LIN {X 6.039,Y -16.044,Z -36.377,A -90.000,B 90.000,C 0.000} C_DIS
LIN {X 6.734,Y -16.027,Z -36.490,A -90.000,B 90.000,C 0.000} C_DIS
LIN {X 7.092,Y -16.027,Z -36.557,A -90.000,B 90.000,C 0.000} C_DIS
LIN {X 7.740,Y -16.017,Z -36.687,A -90.000,B 90.000,C 0.000} C_DIS
LIN {X 9.449,Y -15.968,Z -37.009,A -90.000,B 90.000,C 0.000} C_DIS
LIN {X 9.774,Y -15.964,Z -37.078,A -90.000,B 90.000,C 0.000} C_DIS
LIN {X 10.396,Y -15.956,Z -37.212,A -90.000,B 90.000,C 0.000} C_DIS
LIN {X 11.916,Y -15.912,Z -37.509,A -90.000,B 90.000,C 0.000} C_DIS
LIN {X 12.481,Y -15.903,Z -37.625,A -90.000,B 90.000,C 0.000} C_DIS
LIN {X 13.325,Y -15.897,Z -37.792,A -90.000,B 90.000,C 0.000} C_DIS
LIN {X 14.273,Y -15.872,Z -37.963,A -90.000,B 90.000,C 0.000} C_DIS
LIN {X 14.869,Y -15.862,Z -38.055,A -90.000,B 90.000,C 0.000} C_DIS
LIN {X 16.056,Y -15.855,Z -38.223,A -90.000,B 90.000,C 0.000} C_DIS
LIN {X 16.523,Y -15.850,Z -38.287,A -90.000,B 90.000,C 0.000} C_DIS
LIN {X 16.570,Y -15.848,Z -38.291,A -90.000,B 90.000,C 0.000} C_DIS
LIN {X 16.973,Y -15.845,Z -38.311,A -90.000,B 90.000,C 0.000} C_DIS
LIN {X 17.413,Y -15.859,Z -38.314,A -90.000,B 90.000,C 0.000} C_DIS
LIN {X 18.246,Y -15.862,Z -38.297,A -90.000,B 90.000,C 0.000} C_DIS
LIN {X 19.359,Y -15.901,Z -38.239,A -90.000,B 90.000,C 0.000} C_DIS
LIN {X 20.076,Y -15.912,Z -38.189,A -90.000,B 90.000,C 0.000} C_DIS
LIN {X 20.520,Y -15.912,Z -38.152,A -90.000,B 90.000,C 0.000} C_DIS
LIN {X 21.087,Y -15.918,Z -38.097,A -90.000,B 90.000,C 0.000} C_DIS
LIN {X 21.632,Y -15.923,Z -38.047,A -90.000,B 90.000,C 0.000} C_DIS
LIN {X 22.818,Y -15.923,Z -37.927,A -90.000,B 90.000,C 0.000} C_DIS
LIN {X 23.377,Y -15.913,Z -37.881,A -90.000,B 90.000,C 0.000} C_DIS
LIN {X 23.875,Y -15.906,Z -37.843,A -90.000,B 90.000,C 0.000} C_DIS
LIN {X 24.231,Y -15.897,Z -37.817,A -90.000,B 90.000,C 0.000} C_DIS
LIN {X 24.592,Y -15.885,Z -37.793,A -90.000,B 90.000,C 0.000} C_DIS
LIN {X 25.132,Y -15.871,Z -37.753,A -90.000,B 90.000,C 0.000} C_DIS
LIN {X 26.019,Y -15.831,Z -37.672,A -90.000,B 90.000,C 0.000} C_DIS
LIN {X 26.243,Y -15.824,Z -37.649,A -90.000,B 90.000,C 0.000} C_DIS
LIN {X 26.557,Y -15.821,Z -37.620,A -90.000,B 90.000,C 0.000} C_DIS
LIN {X 26.906,Y -15.809,Z -37.600,A -90.000,B 90.000,C 0.000} C_DIS
LIN {X 27.052,Y -15.798,Z -37.586,A -90.000,B 90.000,C 0.000} C_DIS
LIN {X 27.543,Y -15.770,Z -37.548,A -90.000,B 90.000,C 0.000} C_DIS
LIN {X 27.884,Y -15.754,Z -37.527,A -90.000,B 90.000,C 0.000} C_DIS
LIN {X 28.286,Y -15.743,Z -37.494,A -90.000,B 90.000,C 0.000} C_DIS
LIN {X 28.880,Y -15.723,Z -37.457,A -90.000,B 90.000,C 0.000} C_DIS
LIN {X 29.189,Y -15.702,Z -37.445,A -90.000,B 90.000,C 0.000} C_DIS
LIN {X 29.939,Y -15.655,Z -37.419,A -90.000,B 90.000,C 0.000} C_DIS
LIN {X 30.142,Y -15.646,Z -37.409,A -90.000,B 90.000,C 0.000} C_DIS
LIN {X 30.320,Y -15.634,Z -37.406,A -90.000,B 90.000,C 0.000} C_DIS
LIN {X 30.803,Y -15.614,Z -37.401,A -90.000,B 90.000,C 0.000} C_DIS
LIN {X 31.147,Y -15.605,Z -37.400,A -90.000,B 90.000,C 0.000} C_DIS
LIN {X 31.402,Y -15.589,Z -37.395,A -90.000,B 90.000,C 0.000} C_DIS
LIN {X 32.076,Y -15.550,Z -37.383,A -90.000,B 90.000,C 0.000} C_DIS
LIN {X 32.349,Y -15.534,Z -37.383,A -90.000,B 90.000,C 0.000} C_DIS
LIN {X 33.413,Y -15.503,Z -37.403,A -90.000,B 90.000,C 0.000} C_DIS
LIN {X 33.723,Y -15.486,Z -37.406,A -90.000,B 90.000,C 0.000} C_DIS
LIN {X 34.278,Y -15.462,Z -37.418,A -90.000,B 90.000,C 0.000} C_DIS
LIN {X 34.543,Y -15.456,Z -37.421,A -90.000,B 90.000,C 0.000} C_DIS
LIN {X 34.797,Y -15.450,Z -37.428,A -90.000,B 90.000,C 0.000} C_DIS
LIN {X 35.524,Y -15.428,Z -37.462,A -90.000,B 90.000,C 0.000} C_DIS
LIN {X 36.099,Y -15.416,Z -37.491,A -90.000,B 90.000,C 0.000} C_DIS
LIN {X 36.763,Y -15.397,Z -37.551,A -90.000,B 90.000,C 0.000} C_DIS
LIN {X 37.410,Y -15.387,Z -37.613,A -90.000,B 90.000,C 0.000} C_DIS
LIN {X 37.906,Y -15.374,Z -37.682,A -90.000,B 90.000,C 0.000} C_DIS
LIN {X 38.646,Y -15.360,Z -37.787,A -90.000,B 90.000,C 0.000} C_DIS
LIN {X 39.682,Y -15.341,Z -37.952,A -90.000,B 90.000,C 0.000} C_DIS
LIN {X 40.000,Y -15.341,Z -38.004,A -90.000,B 90.000,C 0.000} C_DIS
LIN {X 40.509,Y -15.338,Z -38.097,A -90.000,B 90.000,C 0.000} C_DIS
LIN {X 41.041,Y -15.331,Z -38.226,A -90.000,B 90.000,C 0.000} C_DIS
LIN {X 42.380,Y -15.317,Z -38.551,A -90.000,B 90.000,C 0.000} C_DIS
LIN {X 43.069,Y -15.313,Z -38.719,A -90.000,B 90.000,C 0.000} C_DIS
LIN {X 43.342,Y -15.313,Z -38.782,A -90.000,B 90.000,C 0.000} C_DIS
LIN {X 43.874,Y -15.312,Z -38.938,A -90.000,B 90.000,C 0.000} C_DIS
LIN {X 45.211,Y -15.309,Z -39.381,A -90.000,B 90.000,C 0.000} C_DIS
LIN {X 46.407,Y -15.308,Z -39.801,A -90.000,B 90.000,C 0.000} C_DIS
LIN {X 46.548,Y -15.315,Z -39.851,A -90.000,B 90.000,C 0.000} C_DIS
LIN {X 46.604,Y -15.308,Z -39.871,A -90.000,B 90.000,C 0.000} C_DIS
LIN {X 47.058,Y -15.309,Z -40.058,A -90.000,B 90.000,C 0.000} C_DIS
LIN {X 49.401,Y -15.308,Z -41.077,A -90.000,B 90.000,C 0.000} C_DIS
LIN {X 49.533,Y -15.308,Z -41.134,A -90.000,B 90.000,C 0.000} C_DIS
LIN {X 49.660,Y -15.308,Z -41.203,A -90.000,B 90.000,C 0.000} C_DIS
LIN {X 49.716,Y -15.308,Z -41.231,A -90.000,B 90.000,C 0.000} C_DIS
LIN {X 50.779,Y -15.308,Z -41.767,A -90.000,B 90.000,C 0.000} C_DIS
LIN {X 51.050,Y -15.308,Z -41.899,A -90.000,B 90.000,C 0.000} C_DIS
LIN {X 51.127,Y -15.308,Z -41.932,A -90.000,B 90.000,C 0.000} C_DIS
LIN {X 51.197,Y -15.308,Z -41.976,A -90.000,B 90.000,C 0.000} C_DIS
LIN {X 51.458,Y -15.308,Z -42.127,A -90.000,B 90.000,C 0.000} C_DIS
LIN {X 52.496,Y -15.308,Z -42.710,A -90.000,B 90.000,C 0.000} C_DIS
LIN {X 52.552,Y -15.308,Z -42.742,A -90.000,B 90.000,C 0.000} C_DIS
LIN {X 53.714,Y -15.307,Z -43.381,A -90.000,B 90.000,C 0.000} C_DIS
LIN {X 54.187,Y -15.306,Z -43.636,A -90.000,B 90.000,C 0.000} C_DIS
LIN {X 54.943,Y -15.302,Z -44.031,A -90.000,B 90.000,C 0.000} C_DIS
LIN {X 55.235,Y -15.300,Z -44.179,A -90.000,B 90.000,C 0.000} C_DIS
LIN {X 55.671,Y -15.295,Z -44.390,A -90.000,B 90.000,C 0.000} C_DIS
LIN {X 56.151,Y -15.273,Z -44.596,A -90.000,B 90.000,C 0.000} C_DIS
LIN {X 56.148,Y -15.270,Z -44.610,A -90.000,B 90.000,C 0.000} C_DIS
LIN {X 56.151,Y -15.268,Z -44.630,A -90.000,B 90.000,C 0.000} C_DIS
LIN {X 56.175,Y -15.267,Z -44.683,A -90.000,B 90.000,C 0.000} C_DIS
LIN {X 56.236,Y -15.266,Z -44.775,A -90.000,B 90.000,C 0.000} C_DIS
LIN {X 56.306,Y -15.267,Z -44.862,A -90.000,B 90.000,C 0.000} C_DIS
LIN {X 56.404,Y -15.268,Z -44.975,A -90.000,B 90.000,C 0.000} C_DIS
LIN {X 56.536,Y -15.269,Z -45.116,A -90.000,B 90.000,C 0.000} C_DIS
LIN {X 56.707,Y -15.272,Z -45.288,A -90.000,B 90.000,C 0.000} C_DIS
LIN {X 56.921,Y -15.275,Z -45.496,A -90.000,B 90.000,C 0.000} C_DIS
LIN {X 57.333,Y -15.281,Z -45.880,A -90.000,B 90.000,C 0.000} C_DIS
LIN {X 57.870,Y -15.289,Z -46.362,A -90.000,B 90.000,C 0.000} C_DIS
LIN {X 58.080,Y -15.293,Z -46.546,A -90.000,B 90.000,C 0.000} C_DIS
LIN {X 58.309,Y -15.296,Z -46.738,A -90.000,B 90.000,C 0.000} C_DIS
LIN {X 58.812,Y -15.304,Z -47.169,A -90.000,B 90.000,C 0.000} C_DIS
LIN {X 59.086,Y -15.308,Z -47.410,A -90.000,B 90.000,C 0.000} C_DIS
LIN {X 59.874,Y -15.321,Z -48.077,A -90.000,B 90.000,C 0.000} C_DIS
LIN {X 59.965,Y -15.308,Z -48.154,A -90.000,B 90.000,C 0.000} C_DIS
LIN {X 60.154,Y -18.803,Z -48.315,A -90.000,B 90.000,C 0.000} C_DIS
LIN {X 60.177,Y -18.801,Z -48.335,A -90.000,B 90.000,C 0.000} C_DIS
LIN {X 60.181,Y -18.797,Z -48.338,A -90.000,B 90.000,C 0.000} C_DIS
LIN {X 60.185,Y -18.774,Z -48.340,A -90.000,B 90.000,C 0.000} C_DIS
LIN {X 60.211,Y -18.708,Z -48.359,A -90.000,B 90.000,C 0.000} C_DIS
LIN {X 60.278,Y -18.515,Z -48.410,A -90.000,B 90.000,C 0.000} C_DIS
LIN {X 60.408,Y -15.308,Z -48.512,A -90.000,B 90.000,C 0.000} C_DIS
LIN {X 61.034,Y -15.309,Z -49.006,A -90.000,B 90.000,C 0.000} C_DIS
LIN {X 61.707,Y -15.310,Z -49.496,A -90.000,B 90.000,C 0.000} C_DIS
LIN {X 62.539,Y -15.313,Z -50.057,A -90.000,B 90.000,C 0.000} C_DIS
LIN {X 63.422,Y -15.320,Z -50.613,A -90.000,B 90.000,C 0.000} C_DIS
LIN {X 63.809,Y -15.325,Z -50.838,A -90.000,B 90.000,C 0.000} C_DIS
LIN {X 64.774,Y -15.332,Z -51.402,A -90.000,B 90.000,C 0.000} C_DIS
LIN {X 65.381,Y -15.337,Z -51.760,A -90.000,B 90.000,C 0.000} C_DIS
LIN {X 65.866,Y -15.341,Z -52.028,A -90.000,B 90.000,C 0.000} C_DIS
LIN {X 66.964,Y -15.343,Z -52.631,A -90.000,B 90.000,C 0.000} C_DIS
LIN {X 67.835,Y -15.347,Z -53.100,A -90.000,B 90.000,C 0.000} C_DIS
LIN {X 70.105,Y -15.348,Z -54.375,A -90.000,B 90.000,C 0.000} C_DIS
LIN {X 72.147,Y -15.347,Z -55.600,A -90.000,B 90.000,C 0.000} C_DIS
LIN {X 72.312,Y -15.348,Z -55.699,A -90.000,B 90.000,C 0.000} C_DIS
LIN {X 74.555,Y -15.349,Z -57.175,A -90.000,B 90.000,C 0.000} C_DIS
LIN {X 74.781,Y -15.352,Z -57.328,A -90.000,B 90.000,C 0.000} C_DIS
LIN {X 75.952,Y -15.356,Z -58.195,A -90.000,B 90.000,C 0.000} C_DIS
LIN {X 76.534,Y -15.359,Z -58.633,A -90.000,B 90.000,C 0.000} C_DIS
LIN {X 76.658,Y -15.359,Z -58.736,A -90.000,B 90.000,C 0.000} C_DIS
LIN {X 77.528,Y -15.366,Z -59.460,A -90.000,B 90.000,C 0.000} C_DIS
LIN {X 78.045,Y -15.370,Z -59.891,A -90.000,B 90.000,C 0.000} C_DIS
LIN {X 78.182,Y -15.370,Z -60.009,A -90.000,B 90.000,C 0.000} C_DIS
LIN {X 78.182,Y -60.000,Z -60.009,A -90.000,B 90.000,C 0.000} C_DIS
LIN {X 98.807,Y -60.000,Z -39.522,A -90.000,B 90.000,C 0.000} C_DIS
LIN {X 98.807,Y -15.308,Z -39.522,A -90.000,B 90.000,C 0.000} C_DIS
LIN {X 98.954,Y -15.308,Z -39.452,A -90.000,B 90.000,C 0.000} C_DIS
LIN {X 98.954,Y -60.000,Z -39.452,A -90.000,B 90.000,C 0.000} C_DIS
LIN {X 117.188,Y -60.000,Z -45.983,A -90.000,B 90.000,C 0.000} C_DIS
LIN {X 117.188,Y -15.308,Z -45.983,A -90.000,B 90.000,C 0.000} C_DIS
LIN {X 117.180,Y -15.308,Z -46.008,A -90.000,B 90.000,C 0.000} C_DIS
LIN {X 117.180,Y -60.000,Z -46.008,A -90.000,B 90.000,C 0.000} C_DIS
LIN {X -92.086,Y -60.000,Z -21.753,A -90.000,B 90.000,C 0.000} C_DIS
LIN {X -92.086,Y -15.308,Z -21.753,A -90.000,B 90.000,C 0.000} C_DIS
LIN {X -91.888,Y -15.383,Z -21.822,A -90.000,B 90.000,C 0.000} C_DIS
LIN {X -91.713,Y -15.437,Z -21.889,A -90.000,B 90.000,C 0.000} C_DIS
LIN {X -91.547,Y -15.487,Z -21.957,A -90.000,B 90.000,C 0.000} C_DIS
LIN {X -91.432,Y -15.522,Z -22.009,A -90.000,B 90.000,C 0.000} C_DIS
LIN {X -91.308,Y -15.555,Z -22.068,A -90.000,B 90.000,C 0.000} C_DIS
LIN {X -91.116,Y -15.602,Z -22.162,A -90.000,B 90.000,C 0.000} C_DIS
LIN {X -90.998,Y -15.635,Z -22.071,A -90.000,B 90.000,C 0.000} C_DIS
LIN {X -90.915,Y -15.658,Z -22.014,A -90.000,B 90.000,C 0.000} C_DIS
LIN {X -90.848,Y -15.675,Z -21.973,A -90.000,B 90.000,C 0.000} C_DIS
LIN {X -90.705,Y -15.711,Z -21.896,A -90.000,B 90.000,C 0.000} C_DIS
LIN {X -90.601,Y -15.737,Z -21.846,A -90.000,B 90.000,C 0.000} C_DIS
LIN {X -90.508,Y -15.760,Z -21.795,A -90.000,B 90.000,C 0.000} C_DIS
LIN {X -90.443,Y -15.772,Z -21.761,A -90.000,B 90.000,C 0.000} C_DIS
LIN {X -90.207,Y -15.808,Z -21.626,A -90.000,B 90.000,C 0.000} C_DIS
LIN {X -89.996,Y -15.833,Z -21.517,A -90.000,B 90.000,C 0.000} C_DIS
LIN {X -89.781,Y -15.852,Z -21.411,A -90.000,B 90.000,C 0.000} C_DIS
LIN {X -89.618,Y -15.868,Z -21.338,A -90.000,B 90.000,C 0.000} C_DIS
LIN {X -89.570,Y -15.872,Z -21.314,A -90.000,B 90.000,C 0.000} C_DIS
LIN {X -89.396,Y -15.862,Z -21.035,A -90.000,B 90.000,C 0.000} C_DIS
LIN {X -89.237,Y -15.854,Z -20.805,A -90.000,B 90.000,C 0.000} C_DIS
LIN {X -89.137,Y -15.841,Z -20.666,A -90.000,B 90.000,C 0.000} C_DIS
LIN {X -89.073,Y -15.829,Z -20.580,A -90.000,B 90.000,C 0.000} C_DIS
LIN {X -88.905,Y -15.795,Z -20.375,A -90.000,B 90.000,C 0.000} C_DIS
LIN {X -88.721,Y -15.747,Z -20.158,A -90.000,B 90.000,C 0.000} C_DIS
LIN {X -88.629,Y -15.719,Z -20.052,A -90.000,B 90.000,C 0.000} C_DIS
LIN {X -88.477,Y -15.662,Z -19.900,A -90.000,B 90.000,C 0.000} C_DIS
LIN {X -88.436,Y -15.647,Z -19.862,A -90.000,B 90.000,C 0.000} C_DIS
LIN {X -88.404,Y -15.624,Z -19.807,A -90.000,B 90.000,C 0.000} C_DIS
LIN {X -88.259,Y -15.535,Z -19.590,A -90.000,B 90.000,C 0.000} C_DIS
LIN {X -88.129,Y -15.439,Z -19.413,A -90.000,B 90.000,C 0.000} C_DIS
LIN {X -88.068,Y -15.399,Z -19.336,A -90.000,B 90.000,C 0.000} C_DIS
LIN {X -87.988,Y -15.346,Z -19.237,A -90.000,B 90.000,C 0.000} C_DIS
LIN {X -87.929,Y -15.308,Z -19.168,A -90.000,B 90.000,C 0.000} C_DIS
LIN {X -87.929,Y -60.000,Z -19.168,A -90.000,B 90.000,C 0.000} C_DIS
LIN {X -116.648,Y -60.000,Z -243.561,A -90.000,B 90.000,C 0.000} C_DIS
LIN {X -116.648,Y -15.666,Z -243.561,A -90.000,B 90.000,C 0.000} C_DIS
LIN {X -116.613,Y -15.603,Z -243.444,A -90.000,B 90.000,C 0.000} C_DIS
LIN {X -116.514,Y -15.450,Z -243.147,A -90.000,B 90.000,C 0.000} C_DIS
LIN {X -116.456,Y -15.375,Z -242.994,A -90.000,B 90.000,C 0.000} C_DIS
LIN {X -116.391,Y -15.308,Z -242.850,A -90.000,B 90.000,C 0.000} C_DIS
LIN {X -116.376,Y -15.293,Z -242.802,A -90.000,B 90.000,C 0.000} C_DIS
LIN {X -116.360,Y -15.273,Z -242.761,A -90.000,B 90.000,C 0.000} C_DIS
LIN {X -116.349,Y -15.254,Z -242.726,A -90.000,B 90.000,C 0.000} C_DIS
LIN {X -116.337,Y -15.221,Z -242.668,A -90.000,B 90.000,C 0.000} C_DIS
LIN {X -116.338,Y -15.193,Z -242.628,A -90.000,B 90.000,C 0.000} C_DIS
LIN {X -116.342,Y -15.182,Z -242.614,A -90.000,B 90.000,C 0.000} C_DIS
LIN {X -116.361,Y -15.161,Z -242.597,A -90.000,B 90.000,C 0.000} C_DIS
LIN {X -116.382,Y -15.146,Z -242.590,A -90.000,B 90.000,C 0.000} C_DIS
LIN {X -116.419,Y -15.130,Z -242.593,A -90.000,B 90.000,C 0.000} C_DIS
LIN {X -116.466,Y -15.118,Z -242.609,A -90.000,B 90.000,C 0.000} C_DIS
LIN {X -116.522,Y -15.110,Z -242.637,A -90.000,B 90.000,C 0.000} C_DIS
LIN {X -116.586,Y -15.105,Z -242.674,A -90.000,B 90.000,C 0.000} C_DIS
LIN {X -116.692,Y -15.103,Z -242.747,A -90.000,B 90.000,C 0.000} C_DIS
LIN {X -116.768,Y -15.105,Z -242.805,A -90.000,B 90.000,C 0.000} C_DIS
LIN {X -116.929,Y -15.117,Z -242.937,A -90.000,B 90.000,C 0.000} C_DIS
LIN {X -117.012,Y -15.126,Z -243.008,A -90.000,B 90.000,C 0.000} C_DIS
LIN {X -117.174,Y -15.148,Z -243.157,A -90.000,B 90.000,C 0.000} C_DIS
LIN {X -117.251,Y -15.161,Z -243.231,A -90.000,B 90.000,C 0.000} C_DIS
LIN {X -117.393,Y -15.189,Z -243.374,A -90.000,B 90.000,C 0.000} C_DIS
LIN {X -117.510,Y -15.218,Z -243.501,A -90.000,B 90.000,C 0.000} C_DIS
LIN {X -117.557,Y -15.233,Z -243.555,A -90.000,B 90.000,C 0.000} C_DIS
LIN {X -117.607,Y -15.254,Z -243.622,A -90.000,B 90.000,C 0.000} C_DIS
LIN {X -117.630,Y -15.273,Z -243.667,A -90.000,B 90.000,C 0.000} C_DIS
LIN {X -117.630,Y -15.284,Z -243.684,A -90.000,B 90.000,C 0.000} C_DIS
LIN {X -117.624,Y -15.290,Z -243.687,A -90.000,B 90.000,C 0.000} C_DIS
LIN {X -117.614,Y -15.295,Z -243.688,A -90.000,B 90.000,C 0.000} C_DIS
LIN {X -117.586,Y -15.302,Z -243.679,A -90.000,B 90.000,C 0.000} C_DIS
LIN {X -117.540,Y -15.308,Z -243.655,A -90.000,B 90.000,C 0.000} C_DIS
LIN {X -117.476,Y -15.312,Z -243.615,A -90.000,B 90.000,C 0.000} C_DIS
LIN {X -117.389,Y -15.308,Z -243.561,A -90.000,B 90.000,C 0.000} C_DIS
LIN {X -115.237,Y -15.308,Z -242.028,A -90.000,B 90.000,C 0.000} C_DIS
LIN {X -113.401,Y -15.308,Z -240.744,A -90.000,B 90.000,C 0.000} C_DIS
LIN {X -107.952,Y -15.308,Z -236.909,A -90.000,B 90.000,C 0.000} C_DIS
LIN {X -105.768,Y -15.308,Z -235.394,A -90.000,B 90.000,C 0.000} C_DIS
LIN {X -100.289,Y -15.308,Z -231.602,A -90.000,B 90.000,C 0.000} C_DIS
LIN {X -98.915,Y -15.308,Z -230.666,A -90.000,B 90.000,C 0.000} C_DIS
LIN {X -92.116,Y -15.308,Z -226.117,A -90.000,B 90.000,C 0.000} C_DIS
LIN {X -91.315,Y -15.308,Z -225.590,A -90.000,B 90.000,C 0.000} C_DIS
LIN {X -84.002,Y -15.308,Z -220.823,A -90.000,B 90.000,C 0.000} C_DIS
LIN {X -78.453,Y -15.308,Z -217.279,A -90.000,B 90.000,C 0.000} C_DIS
LIN {X -75.728,Y -15.308,Z -215.542,A -90.000,B 90.000,C 0.000} C_DIS
LIN {X -71.791,Y -15.308,Z -213.048,A -90.000,B 90.000,C 0.000} C_DIS
LIN {X -67.627,Y -15.308,Z -210.416,A -90.000,B 90.000,C 0.000} C_DIS
LIN {X -65.386,Y -15.308,Z -208.991,A -90.000,B 90.000,C 0.000} C_DIS
LIN {X -60.034,Y -15.308,Z -205.600,A -90.000,B 90.000,C 0.000} C_DIS
LIN {X -59.334,Y -15.308,Z -205.146,A -90.000,B 90.000,C 0.000} C_DIS
LIN {X -56.143,Y -15.308,Z -203.092,A -90.000,B 90.000,C 0.000} C_DIS
LIN {X -53.295,Y -15.308,Z -201.269,A -90.000,B 90.000,C 0.000} C_DIS
LIN {X -49.307,Y -15.308,Z -198.612,A -90.000,B 90.000,C 0.000} C_DIS
LIN {X -47.754,Y -15.308,Z -197.594,A -90.000,B 90.000,C 0.000} C_DIS
LIN {X -43.160,Y -15.308,Z -194.447,A -90.000,B 90.000,C 0.000} C_DIS
LIN {X -41.297,Y -15.308,Z -193.112,A -90.000,B 90.000,C 0.000} C_DIS
LIN {X -39.245,Y -15.308,Z -191.653,A -90.000,B 90.000,C 0.000} C_DIS
LIN {X -39.089,Y -15.308,Z -191.540,A -90.000,B 90.000,C 0.000} C_DIS
LIN {X -35.801,Y -15.308,Z -189.109,A -90.000,B 90.000,C 0.000} C_DIS
LIN {X -32.945,Y -15.308,Z -186.943,A -90.000,B 90.000,C 0.000} C_DIS
LIN {X -32.652,Y -15.308,Z -186.724,A -90.000,B 90.000,C 0.000} C_DIS
LIN {X -29.877,Y -15.308,Z -184.535,A -90.000,B 90.000,C 0.000} C_DIS
LIN {X -27.265,Y -15.308,Z -182.360,A -90.000,B 90.000,C 0.000} C_DIS
LIN {X -24.824,Y -15.308,Z -180.183,A -90.000,B 90.000,C 0.000} C_DIS
LIN {X -22.596,Y -15.308,Z -178.029,A -90.000,B 90.000,C 0.000} C_DIS
LIN {X -20.535,Y -15.308,Z -175.832,A -90.000,B 90.000,C 0.000} C_DIS
LIN {X -18.684,Y -15.308,Z -173.621,A -90.000,B 90.000,C 0.000} C_DIS
LIN {X -18.235,Y -15.308,Z -173.010,A -90.000,B 90.000,C 0.000} C_DIS
LIN {X -16.942,Y -15.308,Z -171.263,A -90.000,B 90.000,C 0.000} C_DIS
LIN {X -15.467,Y -15.308,Z -168.955,A -90.000,B 90.000,C 0.000} C_DIS
LIN {X -14.216,Y -15.308,Z -166.633,A -90.000,B 90.000,C 0.000} C_DIS
LIN {X -14.164,Y -15.308,Z -166.500,A -90.000,B 90.000,C 0.000} C_DIS
LIN {X -13.332,Y -15.308,Z -164.519,A -90.000,B 90.000,C 0.000} C_DIS
LIN {X -13.238,Y -15.308,Z -164.152,A -90.000,B 90.000,C 0.000} C_DIS
LIN {X -12.918,Y -15.308,Z -162.939,A -90.000,B 90.000,C 0.000} C_DIS
LIN {X -12.895,Y -15.308,Z -162.057,A -90.000,B 90.000,C 0.000} C_DIS
LIN {X -13.039,Y -15.308,Z -161.467,A -90.000,B 90.000,C 0.000} C_DIS
LIN {X -13.402,Y -15.308,Z -160.748,A -90.000,B 90.000,C 0.000} C_DIS
LIN {X -14.051,Y -15.308,Z -159.808,A -90.000,B 90.000,C 0.000} C_DIS
LIN {X -14.910,Y -15.308,Z -158.643,A -90.000,B 90.000,C 0.000} C_DIS
LIN {X -15.681,Y -15.308,Z -157.716,A -90.000,B 90.000,C 0.000} C_DIS
LIN {X -15.833,Y -15.308,Z -157.523,A -90.000,B 90.000,C 0.000} C_DIS
LIN {X -17.231,Y -15.308,Z -156.023,A -90.000,B 90.000,C 0.000} C_DIS
LIN {X -17.305,Y -15.308,Z -155.936,A -90.000,B 90.000,C 0.000} C_DIS
LIN {X -19.249,Y -15.308,Z -154.029,A -90.000,B 90.000,C 0.000} C_DIS
LIN {X -21.547,Y -15.308,Z -151.918,A -90.000,B 90.000,C 0.000} C_DIS
LIN {X -21.981,Y -15.308,Z -151.511,A -90.000,B 90.000,C 0.000} C_DIS
LIN {X -25.167,Y -15.308,Z -148.495,A -90.000,B 90.000,C 0.000} C_DIS
LIN {X -25.241,Y -15.308,Z -148.423,A -90.000,B 90.000,C 0.000} C_DIS
LIN {X -28.518,Y -15.308,Z -145.013,A -90.000,B 90.000,C 0.000} C_DIS
LIN {X -28.795,Y -15.308,Z -144.709,A -90.000,B 90.000,C 0.000} C_DIS
LIN {X -28.984,Y -15.308,Z -144.482,A -90.000,B 90.000,C 0.000} C_DIS
LIN {X -31.841,Y -15.308,Z -140.990,A -90.000,B 90.000,C 0.000} C_DIS
LIN {X -32.129,Y -15.308,Z -140.602,A -90.000,B 90.000,C 0.000} C_DIS
LIN {X -34.151,Y -15.308,Z -137.405,A -90.000,B 90.000,C 0.000} C_DIS
LIN {X -34.657,Y -15.308,Z -136.618,A -90.000,B 90.000,C 0.000} C_DIS
LIN {X -34.903,Y -15.308,Z -136.203,A -90.000,B 90.000,C 0.000} C_DIS
LIN {X -36.290,Y -15.308,Z -133.519,A -90.000,B 90.000,C 0.000} C_DIS
LIN {X -36.962,Y -15.308,Z -132.232,A -90.000,B 90.000,C 0.000} C_DIS
LIN {X -37.164,Y -15.308,Z -131.794,A -90.000,B 90.000,C 0.000} C_DIS
LIN {X -38.019,Y -15.308,Z -129.863,A -90.000,B 90.000,C 0.000} C_DIS
LIN {X -38.802,Y -15.308,Z -128.109,A -90.000,B 90.000,C 0.000} C_DIS
LIN {X -39.251,Y -15.308,Z -126.997,A -90.000,B 90.000,C 0.000} C_DIS
LIN {X -40.072,Y -15.308,Z -124.975,A -90.000,B 90.000,C 0.000} C_DIS
LIN {X -41.025,Y -15.308,Z -122.667,A -90.000,B 90.000,C 0.000} C_DIS
LIN {X -41.568,Y -15.308,Z -121.483,A -90.000,B 90.000,C 0.000} C_DIS
LIN {X -41.695,Y -15.308,Z -121.225,A -90.000,B 90.000,C 0.000} C_DIS
LIN {X -42.223,Y -15.308,Z -120.307,A -90.000,B 90.000,C 0.000} C_DIS
LIN {X -42.435,Y -15.308,Z -119.959,A -90.000,B 90.000,C 0.000} C_DIS
LIN {X -43.086,Y -15.308,Z -119.039,A -90.000,B 90.000,C 0.000} C_DIS
LIN {X -43.497,Y -15.308,Z -118.478,A -90.000,B 90.000,C 0.000} C_DIS
LIN {X -44.840,Y -15.308,Z -116.818,A -90.000,B 90.000,C 0.000} C_DIS
LIN {X -45.304,Y -15.308,Z -116.239,A -90.000,B 90.000,C 0.000} C_DIS
LIN {X -47.568,Y -15.308,Z -113.521,A -90.000,B 90.000,C 0.000} C_DIS
LIN {X -50.011,Y -15.308,Z -110.539,A -90.000,B 90.000,C 0.000} C_DIS
LIN {X -51.120,Y -15.308,Z -109.126,A -90.000,B 90.000,C 0.000} C_DIS
LIN {X -52.562,Y -15.308,Z -107.296,A -90.000,B 90.000,C 0.000} C_DIS
LIN {X -55.328,Y -15.308,Z -103.554,A -90.000,B 90.000,C 0.000} C_DIS
LIN {X -56.973,Y -15.308,Z -101.251,A -90.000,B 90.000,C 0.000} C_DIS
LIN {X -58.587,Y -15.308,Z -99.016,A -90.000,B 90.000,C 0.000} C_DIS
LIN {X -59.885,Y -15.308,Z -97.233,A -90.000,B 90.000,C 0.000} C_DIS
LIN {X -61.927,Y -15.308,Z -94.532,A -90.000,B 90.000,C 0.000} C_DIS
LIN {X -62.921,Y -15.308,Z -93.319,A -90.000,B 90.000,C 0.000} C_DIS
LIN {X -63.877,Y -15.308,Z -92.127,A -90.000,B 90.000,C 0.000} C_DIS
LIN {X -64.860,Y -15.308,Z -91.036,A -90.000,B 90.000,C 0.000} C_DIS
LIN {X -65.598,Y -15.308,Z -90.186,A -90.000,B 90.000,C 0.000} C_DIS
LIN {X -66.357,Y -15.308,Z -89.434,A -90.000,B 90.000,C 0.000} C_DIS
LIN {X -67.270,Y -15.308,Z -88.483,A -90.000,B 90.000,C 0.000} C_DIS
LIN {X -68.319,Y -15.308,Z -87.558,A -90.000,B 90.000,C 0.000} C_DIS
LIN {X -69.110,Y -15.308,Z -86.821,A -90.000,B 90.000,C 0.000} C_DIS
LIN {X -69.918,Y -15.308,Z -86.149,A -90.000,B 90.000,C 0.000} C_DIS
LIN {X -70.867,Y -15.308,Z -85.391,A -90.000,B 90.000,C 0.000} C_DIS
LIN {X -71.643,Y -15.308,Z -84.802,A -90.000,B 90.000,C 0.000} C_DIS
LIN {X -73.034,Y -15.308,Z -83.787,A -90.000,B 90.000,C 0.000} C_DIS
LIN {X -73.968,Y -15.308,Z -83.142,A -90.000,B 90.000,C 0.000} C_DIS
LIN {X -74.795,Y -15.308,Z -82.588,A -90.000,B 90.000,C 0.000} C_DIS
LIN {X -75.787,Y -15.308,Z -81.979,A -90.000,B 90.000,C 0.000} C_DIS
LIN {X -76.836,Y -15.308,Z -81.337,A -90.000,B 90.000,C 0.000} C_DIS
LIN {X -78.172,Y -15.308,Z -80.600,A -90.000,B 90.000,C 0.000} C_DIS
LIN {X -79.737,Y -15.308,Z -79.776,A -90.000,B 90.000,C 0.000} C_DIS
LIN {X -80.389,Y -15.308,Z -79.422,A -90.000,B 90.000,C 0.000} C_DIS
LIN {X -81.547,Y -15.308,Z -78.791,A -90.000,B 90.000,C 0.000} C_DIS
LIN {X -81.922,Y -15.308,Z -78.581,A -90.000,B 90.000,C 0.000} C_DIS
LIN {X -82.041,Y -15.308,Z -78.501,A -90.000,B 90.000,C 0.000} C_DIS
LIN {X -83.191,Y -15.308,Z -77.779,A -90.000,B 90.000,C 0.000} C_DIS
LIN {X -83.548,Y -15.308,Z -77.541,A -90.000,B 90.000,C 0.000} C_DIS
LIN {X -83.614,Y -15.308,Z -77.499,A -90.000,B 90.000,C 0.000} C_DIS
LIN {X -83.687,Y -15.308,Z -77.446,A -90.000,B 90.000,C 0.000} C_DIS
LIN {X -84.755,Y -15.308,Z -76.642,A -90.000,B 90.000,C 0.000} C_DIS
LIN {X -85.186,Y -15.308,Z -76.299,A -90.000,B 90.000,C 0.000} C_DIS
LIN {X -86.321,Y -15.308,Z -75.357,A -90.000,B 90.000,C 0.000} C_DIS
LIN {X -87.009,Y -15.308,Z -74.773,A -90.000,B 90.000,C 0.000} C_DIS
LIN {X -87.618,Y -15.308,Z -74.268,A -90.000,B 90.000,C 0.000} C_DIS
LIN {X -87.941,Y -15.308,Z -74.029,A -90.000,B 90.000,C 0.000} C_DIS
LIN {X -88.343,Y -15.308,Z -73.713,A -90.000,B 90.000,C 0.000} C_DIS
LIN {X -88.766,Y -15.308,Z -73.430,A -90.000,B 90.000,C 0.000} C_DIS
LIN {X -88.994,Y -15.308,Z -73.263,A -90.000,B 90.000,C 0.000} C_DIS
LIN {X -89.525,Y -15.308,Z -72.943,A -90.000,B 90.000,C 0.000} C_DIS
LIN {X -89.590,Y -15.308,Z -72.912,A -90.000,B 90.000,C 0.000} C_DIS
LIN {X -89.646,Y -15.308,Z -72.882,A -90.000,B 90.000,C 0.000} C_DIS
LIN {X -90.088,Y -15.308,Z -72.650,A -90.000,B 90.000,C 0.000} C_DIS
LIN {X -90.570,Y -15.308,Z -72.448,A -90.000,B 90.000,C 0.000} C_DIS
LIN {X -90.858,Y -15.308,Z -72.316,A -90.000,B 90.000,C 0.000} C_DIS
LIN {X -91.444,Y -15.308,Z -72.093,A -90.000,B 90.000,C 0.000} C_DIS
LIN {X -92.043,Y -15.308,Z -71.877,A -90.000,B 90.000,C 0.000} C_DIS
LIN {X -92.532,Y -15.308,Z -71.728,A -90.000,B 90.000,C 0.000} C_DIS
LIN {X -93.086,Y -15.308,Z -71.530,A -90.000,B 90.000,C 0.000} C_DIS
LIN {X -93.888,Y -15.308,Z -71.305,A -90.000,B 90.000,C 0.000} C_DIS
LIN {X -94.287,Y -15.308,Z -71.174,A -90.000,B 90.000,C 0.000} C_DIS
LIN {X -94.391,Y -15.308,Z -71.155,A -90.000,B 90.000,C 0.000} C_DIS
LIN {X -94.652,Y -15.308,Z -71.078,A -90.000,B 90.000,C 0.000} C_DIS
LIN {X -95.192,Y -15.308,Z -70.980,A -90.000,B 90.000,C 0.000} C_DIS
LIN {X -95.452,Y -15.308,Z -70.918,A -90.000,B 90.000,C 0.000} C_DIS
LIN {X -96.402,Y -15.308,Z -70.652,A -90.000,B 90.000,C 0.000} C_DIS
LIN {X -96.813,Y -15.308,Z -70.531,A -90.000,B 90.000,C 0.000} C_DIS
LIN {X -97.204,Y -15.308,Z -70.390,A -90.000,B 90.000,C 0.000} C_DIS
LIN {X -97.470,Y -15.308,Z -70.331,A -90.000,B 90.000,C 0.000} C_DIS
LIN {X -97.877,Y -15.308,Z -70.212,A -90.000,B 90.000,C 0.000} C_DIS
LIN {X -98.286,Y -15.308,Z -70.036,A -90.000,B 90.000,C 0.000} C_DIS
LIN {X -98.901,Y -15.308,Z -69.833,A -90.000,B 90.000,C 0.000} C_DIS
LIN {X -99.387,Y -15.308,Z -69.625,A -90.000,B 90.000,C 0.000} C_DIS
LIN {X -99.576,Y -15.308,Z -69.516,A -90.000,B 90.000,C 0.000} C_DIS
LIN {X -100.478,Y -15.308,Z -69.076,A -90.000,B 90.000,C 0.000} C_DIS
LIN {X -100.930,Y -15.308,Z -68.811,A -90.000,B 90.000,C 0.000} C_DIS
LIN {X -101.280,Y -15.308,Z -68.551,A -90.000,B 90.000,C 0.000} C_DIS
LIN {X -102.025,Y -15.308,Z -68.035,A -90.000,B 90.000,C 0.000} C_DIS
LIN {X -102.496,Y -15.308,Z -67.685,A -90.000,B 90.000,C 0.000} C_DIS
LIN {X -103.303,Y -15.308,Z -66.929,A -90.000,B 90.000,C 0.000} C_DIS
LIN {X -103.460,Y -15.308,Z -66.780,A -90.000,B 90.000,C 0.000} C_DIS
LIN {X -104.066,Y -15.308,Z -66.172,A -90.000,B 90.000,C 0.000} C_DIS
LIN {X -104.374,Y -15.308,Z -65.825,A -90.000,B 90.000,C 0.000} C_DIS
LIN {X -105.252,Y -15.308,Z -64.773,A -90.000,B 90.000,C 0.000} C_DIS
LIN {X -105.502,Y -15.308,Z -64.437,A -90.000,B 90.000,C 0.000} C_DIS
LIN {X -105.663,Y -15.308,Z -64.191,A -90.000,B 90.000,C 0.000} C_DIS
LIN {X -105.942,Y -15.308,Z -63.748,A -90.000,B 90.000,C 0.000} C_DIS
LIN {X -106.247,Y -15.308,Z -63.249,A -90.000,B 90.000,C 0.000} C_DIS
LIN {X -106.464,Y -15.308,Z -62.881,A -90.000,B 90.000,C 0.000} C_DIS
LIN {X -106.848,Y -15.308,Z -62.209,A -90.000,B 90.000,C 0.000} C_DIS
LIN {X -107.351,Y -15.308,Z -61.238,A -90.000,B 90.000,C 0.000} C_DIS
LIN {X -107.596,Y -15.308,Z -60.653,A -90.000,B 90.000,C 0.000} C_DIS
LIN {X -107.676,Y -15.308,Z -60.452,A -90.000,B 90.000,C 0.000} C_DIS
LIN {X -107.925,Y -15.308,Z -59.786,A -90.000,B 90.000,C 0.000} C_DIS
LIN {X -108.175,Y -15.308,Z -59.057,A -90.000,B 90.000,C 0.000} C_DIS
LIN {X -108.232,Y -15.308,Z -58.865,A -90.000,B 90.000,C 0.000} C_DIS
LIN {X -108.340,Y -15.308,Z -58.477,A -90.000,B 90.000,C 0.000} C_DIS
LIN {X -108.517,Y -15.308,Z -57.790,A -90.000,B 90.000,C 0.000} C_DIS
LIN {X -108.694,Y -15.308,Z -57.036,A -90.000,B 90.000,C 0.000} C_DIS
LIN {X -108.705,Y -15.308,Z -56.978,A -90.000,B 90.000,C 0.000} C_DIS
LIN {X -108.794,Y -15.308,Z -56.618,A -90.000,B 90.000,C 0.000} C_DIS
LIN {X -108.994,Y -15.308,Z -56.353,A -90.000,B 90.000,C 0.000} C_DIS
LIN {X -109.232,Y -15.308,Z -56.034,A -90.000,B 90.000,C 0.000} C_DIS
LIN {X -109.310,Y -15.308,Z -55.934,A -90.000,B 90.000,C 0.000} C_DIS
LIN {X -109.476,Y -15.308,Z -55.711,A -90.000,B 90.000,C 0.000} C_DIS
LIN {X -109.604,Y -15.308,Z -55.550,A -90.000,B 90.000,C 0.000} C_DIS
LIN {X -109.701,Y -15.308,Z -55.423,A -90.000,B 90.000,C 0.000} C_DIS
LIN {X -109.823,Y -15.308,Z -55.268,A -90.000,B 90.000,C 0.000} C_DIS
LIN {X -109.916,Y -15.308,Z -55.134,A -90.000,B 90.000,C 0.000} C_DIS
LIN {X -109.982,Y -15.308,Z -55.044,A -90.000,B 90.000,C 0.000} C_DIS
LIN {X -110.100,Y -15.308,Z -54.874,A -90.000,B 90.000,C 0.000} C_DIS
LIN {X -110.245,Y -15.308,Z -54.674,A -90.000,B 90.000,C 0.000} C_DIS
LIN {X -110.337,Y -15.308,Z -54.542,A -90.000,B 90.000,C 0.000} C_DIS
LIN {X -110.708,Y -15.308,Z -53.981,A -90.000,B 90.000,C 0.000} C_DIS
LIN {X -110.962,Y -15.308,Z -53.565,A -90.000,B 90.000,C 0.000} C_DIS
LIN {X -111.206,Y -15.308,Z -53.096,A -90.000,B 90.000,C 0.000} C_DIS
LIN {X -111.406,Y -15.308,Z -52.674,A -90.000,B 90.000,C 0.000} C_DIS
LIN {X -111.446,Y -15.308,Z -52.585,A -90.000,B 90.000,C 0.000} C_DIS
LIN {X -111.625,Y -15.308,Z -52.147,A -90.000,B 90.000,C 0.000} C_DIS
LIN {X -111.669,Y -15.308,Z -52.024,A -90.000,B 90.000,C 0.000} C_DIS
LIN {X -111.810,Y -15.308,Z -51.591,A -90.000,B 90.000,C 0.000} C_DIS
LIN {X -111.903,Y -15.308,Z -51.154,A -90.000,B 90.000,C 0.000} C_DIS
LIN {X -111.987,Y -15.308,Z -50.742,A -90.000,B 90.000,C 0.000} C_DIS
LIN {X -112.049,Y -15.308,Z -50.261,A -90.000,B 90.000,C 0.000} C_DIS
LIN {X -112.088,Y -15.308,Z -49.822,A -90.000,B 90.000,C 0.000} C_DIS
LIN {X -112.078,Y -15.308,Z -49.381,A -90.000,B 90.000,C 0.000} C_DIS
LIN {X -112.070,Y -15.308,Z -49.209,A -90.000,B 90.000,C 0.000} C_DIS
LIN {X -112.063,Y -15.308,Z -49.133,A -90.000,B 90.000,C 0.000} C_DIS
LIN {X -112.007,Y -15.308,Z -48.713,A -90.000,B 90.000,C 0.000} C_DIS
LIN {X -111.939,Y -15.308,Z -48.279,A -90.000,B 90.000,C 0.000} C_DIS
LIN {X -111.834,Y -15.308,Z -47.869,A -90.000,B 90.000,C 0.000} C_DIS
LIN {X -111.692,Y -15.308,Z -47.455,A -90.000,B 90.000,C 0.000} C_DIS
LIN {X -111.530,Y -15.308,Z -47.039,A -90.000,B 90.000,C 0.000} C_DIS
LIN {X -111.504,Y -15.308,Z -46.979,A -90.000,B 90.000,C 0.000} C_DIS
LIN {X -111.330,Y -15.308,Z -46.616,A -90.000,B 90.000,C 0.000} C_DIS
LIN {X -111.129,Y -15.308,Z -46.226,A -90.000,B 90.000,C 0.000} C_DIS
LIN {X -111.074,Y -15.308,Z -46.132,A -90.000,B 90.000,C 0.000} C_DIS
LIN {X -111.119,Y -15.308,Z -46.053,A -90.000,B 90.000,C 0.000} C_DIS
LIN {X -111.352,Y -15.308,Z -45.633,A -90.000,B 90.000,C 0.000} C_DIS
LIN {X -111.487,Y -15.308,Z -45.370,A -90.000,B 90.000,C 0.000} C_DIS
LIN {X -111.845,Y -15.308,Z -44.612,A -90.000,B 90.000,C 0.000} C_DIS
LIN {X -112.142,Y -15.308,Z -43.916,A -90.000,B 90.000,C 0.000} C_DIS
LIN {X -112.314,Y -15.308,Z -43.500,A -90.000,B 90.000,C 0.000} C_DIS
LIN {X -112.357,Y -15.308,Z -43.382,A -90.000,B 90.000,C 0.000} C_DIS
LIN {X -112.607,Y -15.308,Z -42.619,A -90.000,B 90.000,C 0.000} C_DIS
LIN {X -112.724,Y -15.308,Z -42.185,A -90.000,B 90.000,C 0.000} C_DIS
LIN {X -112.822,Y -15.308,Z -41.754,A -90.000,B 90.000,C 0.000} C_DIS
LIN {X -112.993,Y -15.308,Z -40.920,A -90.000,B 90.000,C 0.000} C_DIS
LIN {X -113.043,Y -15.308,Z -40.549,A -90.000,B 90.000,C 0.000} C_DIS
LIN {X -113.082,Y -15.308,Z -40.110,A -90.000,B 90.000,C 0.000} C_DIS
LIN {X -113.095,Y -15.308,Z -39.772,A -90.000,B 90.000,C 0.000} C_DIS
LIN {X -113.080,Y -15.308,Z -39.077,A -90.000,B 90.000,C 0.000} C_DIS
LIN {X -113.065,Y -15.308,Z -38.767,A -90.000,B 90.000,C 0.000} C_DIS
LIN {X -112.986,Y -15.308,Z -38.181,A -90.000,B 90.000,C 0.000} C_DIS
LIN {X -112.967,Y -15.308,Z -38.057,A -90.000,B 90.000,C 0.000} C_DIS
LIN {X -112.903,Y -15.308,Z -37.781,A -90.000,B 90.000,C 0.000} C_DIS
LIN {X -112.790,Y -15.308,Z -37.339,A -90.000,B 90.000,C 0.000} C_DIS
LIN {X -112.766,Y -15.308,Z -37.254,A -90.000,B 90.000,C 0.000} C_DIS
LIN {X -112.686,Y -15.308,Z -36.995,A -90.000,B 90.000,C 0.000} C_DIS
LIN {X -112.460,Y -15.308,Z -36.380,A -90.000,B 90.000,C 0.000} C_DIS
LIN {X -112.439,Y -15.308,Z -36.330,A -90.000,B 90.000,C 0.000} C_DIS
LIN {X -112.325,Y -15.308,Z -36.088,A -90.000,B 90.000,C 0.000} C_DIS
LIN {X -112.138,Y -15.308,Z -35.725,A -90.000,B 90.000,C 0.000} C_DIS
LIN {X -111.987,Y -15.308,Z -35.475,A -90.000,B 90.000,C 0.000} C_DIS
LIN {X -111.760,Y -15.308,Z -35.142,A -90.000,B 90.000,C 0.000} C_DIS
LIN {X -111.572,Y -15.308,Z -34.908,A -90.000,B 90.000,C 0.000} C_DIS
LIN {X -111.306,Y -15.308,Z -34.606,A -90.000,B 90.000,C 0.000} C_DIS
LIN {X -111.071,Y -15.308,Z -34.395,A -90.000,B 90.000,C 0.000} C_DIS
LIN {X -110.771,Y -15.308,Z -34.131,A -90.000,B 90.000,C 0.000} C_DIS
LIN {X -110.519,Y -15.308,Z -33.934,A -90.000,B 90.000,C 0.000} C_DIS
LIN {X -110.298,Y -15.308,Z -33.756,A -90.000,B 90.000,C 0.000} C_DIS
LIN {X -110.270,Y -15.308,Z -33.730,A -90.000,B 90.000,C 0.000} C_DIS
LIN {X -110.201,Y -15.308,Z -33.650,A -90.000,B 90.000,C 0.000} C_DIS
LIN {X -109.643,Y -15.308,Z -32.941,A -90.000,B 90.000,C 0.000} C_DIS
LIN {X -109.389,Y -15.308,Z -32.642,A -90.000,B 90.000,C 0.000} C_DIS
LIN {X -109.057,Y -15.308,Z -32.259,A -90.000,B 90.000,C 0.000} C_DIS
LIN {X -108.659,Y -15.308,Z -31.866,A -90.000,B 90.000,C 0.000} C_DIS
LIN {X -108.379,Y -15.308,Z -31.611,A -90.000,B 90.000,C 0.000} C_DIS
LIN {X -108.263,Y -15.308,Z -31.510,A -90.000,B 90.000,C 0.000} C_DIS
LIN {X -107.942,Y -15.308,Z -31.225,A -90.000,B 90.000,C 0.000} C_DIS
LIN {X -107.480,Y -15.308,Z -30.845,A -90.000,B 90.000,C 0.000} C_DIS
LIN {X -106.546,Y -15.308,Z -30.110,A -90.000,B 90.000,C 0.000} C_DIS
LIN {X -106.050,Y -15.308,Z -29.761,A -90.000,B 90.000,C 0.000} C_DIS
LIN {X -105.738,Y -15.308,Z -29.546,A -90.000,B 90.000,C 0.000} C_DIS
LIN {X -105.159,Y -15.308,Z -29.209,A -90.000,B 90.000,C 0.000} C_DIS
LIN {X -104.820,Y -15.308,Z -29.035,A -90.000,B 90.000,C 0.000} C_DIS
LIN {X -104.213,Y -15.308,Z -28.771,A -90.000,B 90.000,C 0.000} C_DIS
LIN {X -104.140,Y -15.308,Z -28.737,A -90.000,B 90.000,C 0.000} C_DIS
LIN {X -103.980,Y -15.308,Z -28.672,A -90.000,B 90.000,C 0.000} C_DIS
LIN {X -103.602,Y -15.308,Z -28.533,A -90.000,B 90.000,C 0.000} C_DIS
LIN {X -103.367,Y -15.308,Z -28.457,A -90.000,B 90.000,C 0.000} C_DIS
LIN {X -102.814,Y -15.308,Z -28.261,A -90.000,B 90.000,C 0.000} C_DIS
LIN {X -102.645,Y -15.308,Z -28.206,A -90.000,B 90.000,C 0.000} C_DIS
LIN {X -102.133,Y -15.308,Z -28.049,A -90.000,B 90.000,C 0.000} C_DIS
LIN {X -101.951,Y -15.308,Z -27.985,A -90.000,B 90.000,C 0.000} C_DIS
LIN {X -101.708,Y -15.308,Z -27.521,A -90.000,B 90.000,C 0.000} C_DIS
LIN {X -101.545,Y -15.308,Z -27.257,A -90.000,B 90.000,C 0.000} C_DIS
LIN {X -101.179,Y -15.308,Z -26.730,A -90.000,B 90.000,C 0.000} C_DIS
LIN {X -101.099,Y -15.308,Z -26.619,A -90.000,B 90.000,C 0.000} C_DIS
LIN {X -100.606,Y -15.308,Z -25.981,A -90.000,B 90.000,C 0.000} C_DIS
LIN {X -100.353,Y -15.308,Z -25.679,A -90.000,B 90.000,C 0.000} C_DIS
LIN {X -99.943,Y -15.308,Z -25.213,A -90.000,B 90.000,C 0.000} C_DIS
LIN {X -99.748,Y -15.308,Z -25.016,A -90.000,B 90.000,C 0.000} C_DIS
LIN {X -99.678,Y -15.308,Z -24.937,A -90.000,B 90.000,C 0.000} C_DIS
LIN {X -99.530,Y -15.308,Z -24.804,A -90.000,B 90.000,C 0.000} C_DIS
LIN {X -99.435,Y -15.308,Z -24.710,A -90.000,B 90.000,C 0.000} C_DIS
LIN {X -99.119,Y -15.308,Z -24.427,A -90.000,B 90.000,C 0.000} C_DIS
LIN {X -98.889,Y -15.308,Z -24.238,A -90.000,B 90.000,C 0.000} C_DIS
LIN {X -98.819,Y -15.308,Z -24.185,A -90.000,B 90.000,C 0.000} C_DIS
LIN {X -98.301,Y -15.308,Z -23.820,A -90.000,B 90.000,C 0.000} C_DIS
LIN {X -98.068,Y -15.308,Z -23.668,A -90.000,B 90.000,C 0.000} C_DIS
LIN {X -97.704,Y -15.308,Z -23.471,A -90.000,B 90.000,C 0.000} C_DIS
LIN {X -97.482,Y -15.308,Z -23.369,A -90.000,B 90.000,C 0.000} C_DIS
LIN {X -97.069,Y -15.308,Z -23.205,A -90.000,B 90.000,C 0.000} C_DIS
LIN {X -96.674,Y -15.308,Z -23.093,A -90.000,B 90.000,C 0.000} C_DIS
LIN {X -96.615,Y -15.308,Z -23.082,A -90.000,B 90.000,C 0.000} C_DIS
LIN {X -96.428,Y -15.308,Z -23.032,A -90.000,B 90.000,C 0.000} C_DIS
LIN {X -95.995,Y -15.308,Z -22.951,A -90.000,B 90.000,C 0.000} C_DIS
LIN {X -95.555,Y -15.308,Z -22.918,A -90.000,B 90.000,C 0.000} C_DIS
LIN {X -95.448,Y -15.308,Z -22.920,A -90.000,B 90.000,C 0.000} C_DIS
LIN {X -95.122,Y -15.308,Z -22.933,A -90.000,B 90.000,C 0.000} C_DIS
LIN {X -95.004,Y -15.308,Z -22.943,A -90.000,B 90.000,C 0.000} C_DIS
LIN {X -94.422,Y -15.308,Z -23.006,A -90.000,B 90.000,C 0.000} C_DIS
LIN {X -93.975,Y -15.308,Z -23.096,A -90.000,B 90.000,C 0.000} C_DIS
LIN {X -93.510,Y -15.308,Z -23.236,A -90.000,B 90.000,C 0.000} C_DIS
LIN {X -93.070,Y -15.308,Z -23.392,A -90.000,B 90.000,C 0.000} C_DIS
LIN {X -92.574,Y -15.308,Z -23.619,A -90.000,B 90.000,C 0.000} C_DIS
LIN {X -91.868,Y -15.308,Z -23.976,A -90.000,B 90.000,C 0.000} C_DIS
LIN {X -91.771,Y -15.308,Z -24.019,A -90.000,B 90.000,C 0.000} C_DIS
LIN {X -91.356,Y -15.308,Z -24.237,A -90.000,B 90.000,C 0.000} C_DIS
LIN {X -91.053,Y -15.308,Z -24.365,A -90.000,B 90.000,C 0.000} C_DIS
LIN {X -90.898,Y -15.308,Z -24.418,A -90.000,B 90.000,C 0.000} C_DIS
LIN {X -90.600,Y -15.308,Z -24.488,A -90.000,B 90.000,C 0.000} C_DIS
LIN {X -90.167,Y -15.308,Z -24.550,A -90.000,B 90.000,C 0.000} C_DIS
LIN {X -89.768,Y -15.308,Z -24.579,A -90.000,B 90.000,C 0.000} C_DIS
LIN {X -89.304,Y -15.308,Z -24.582,A -90.000,B 90.000,C 0.000} C_DIS
LIN {X -89.053,Y -15.308,Z -24.566,A -90.000,B 90.000,C 0.000} C_DIS
LIN {X -90.014,Y -15.308,Z -24.316,A -90.000,B 90.000,C 0.000} C_DIS
LIN {X -90.107,Y -15.308,Z -24.280,A -90.000,B 90.000,C 0.000} C_DIS
LIN {X -90.317,Y -15.308,Z -24.189,A -90.000,B 90.000,C 0.000} C_DIS
LIN {X -90.530,Y -15.308,Z -24.090,A -90.000,B 90.000,C 0.000} C_DIS
LIN {X -90.799,Y -15.308,Z -23.919,A -90.000,B 90.000,C 0.000} C_DIS
LIN {X -91.185,Y -15.308,Z -23.646,A -90.000,B 90.000,C 0.000} C_DIS
LIN {X -91.412,Y -15.308,Z -23.443,A -90.000,B 90.000,C 0.000} C_DIS
LIN {X -91.593,Y -15.308,Z -23.267,A -90.000,B 90.000,C 0.000} C_DIS
LIN {X -91.675,Y -15.308,Z -23.168,A -90.000,B 90.000,C 0.000} C_DIS
LIN {X -91.847,Y -15.308,Z -22.947,A -90.000,B 90.000,C 0.000} C_DIS
LIN {X -91.980,Y -15.308,Z -22.699,A -90.000,B 90.000,C 0.000} C_DIS
LIN {X -92.067,Y -15.308,Z -22.430,A -90.000,B 90.000,C 0.000} C_DIS
LIN {X -92.105,Y -15.308,Z -22.151,A -90.000,B 90.000,C 0.000} C_DIS
LIN {X -92.105,Y -15.308,Z -22.083,A -90.000,B 90.000,C 0.000} C_DIS
LIN {X -92.093,Y -15.308,Z -21.801,A -90.000,B 90.000,C 0.000} C_DIS
LIN {X -92.058,Y -15.308,Z -21.568,A -90.000,B 90.000,C 0.000} C_DIS
LIN {X -91.997,Y -15.308,Z -21.293,A -90.000,B 90.000,C 0.000} C_DIS
LIN {X -91.866,Y -15.308,Z -20.982,A -90.000,B 90.000,C 0.000} C_DIS
LIN {X -91.711,Y -15.308,Z -20.740,A -90.000,B 90.000,C 0.000} C_DIS
LIN {X -91.675,Y -15.308,Z -20.699,A -90.000,B 90.000,C 0.000} C_DIS
LIN {X -91.516,Y -15.308,Z -20.527,A -90.000,B 90.000,C 0.000} C_DIS
LIN {X -91.204,Y -15.308,Z -20.237,A -90.000,B 90.000,C 0.000} C_DIS
LIN {X -90.959,Y -15.308,Z -20.032,A -90.000,B 90.000,C 0.000} C_DIS
LIN {X -90.692,Y -15.308,Z -19.856,A -90.000,B 90.000,C 0.000} C_DIS
LIN {X -90.511,Y -15.308,Z -19.747,A -90.000,B 90.000,C 0.000} C_DIS
LIN {X -90.406,Y -15.308,Z -19.691,A -90.000,B 90.000,C 0.000} C_DIS
LIN {X -90.110,Y -15.308,Z -19.572,A -90.000,B 90.000,C 0.000} C_DIS
LIN {X -89.129,Y -15.308,Z -19.263,A -90.000,B 90.000,C 0.000} C_DIS
LIN {X -88.928,Y -15.308,Z -19.217,A -90.000,B 90.000,C 0.000} C_DIS
LIN {X -88.807,Y -15.308,Z -19.191,A -90.000,B 90.000,C 0.000} C_DIS
LIN {X -88.477,Y -15.308,Z -19.168,A -90.000,B 90.000,C 0.000} C_DIS
LIN {X -87.394,Y -15.308,Z -19.167,A -90.000,B 90.000,C 0.000} C_DIS
LIN {X -87.061,Y -15.308,Z -19.194,A -90.000,B 90.000,C 0.000} C_DIS
LIN {X -87.002,Y -15.308,Z -19.206,A -90.000,B 90.000,C 0.000} C_DIS
LIN {X -86.659,Y -15.308,Z -19.282,A -90.000,B 90.000,C 0.000} C_DIS
LIN {X -86.250,Y -15.308,Z -19.438,A -90.000,B 90.000,C 0.000} C_DIS
LIN {X -85.766,Y -15.308,Z -19.636,A -90.000,B 90.000,C 0.000} C_DIS
LIN {X -85.755,Y -15.308,Z -19.556,A -90.000,B 90.000,C 0.000} C_DIS
LIN {X -85.646,Y -15.308,Z -19.129,A -90.000,B 90.000,C 0.000} C_DIS
LIN {X -85.547,Y -15.308,Z -18.843,A -90.000,B 90.000,C 0.000} C_DIS
LIN {X -85.390,Y -15.308,Z -18.431,A -90.000,B 90.000,C 0.000} C_DIS
LIN {X -85.191,Y -15.308,Z -18.048,A -90.000,B 90.000,C 0.000} C_DIS
LIN {X -85.016,Y -15.308,Z -17.769,A -90.000,B 90.000,C 0.000} C_DIS
LIN {X -84.776,Y -15.308,Z -17.414,A -90.000,B 90.000,C 0.000} C_DIS
LIN {X -84.490,Y -15.308,Z -17.078,A -90.000,B 90.000,C 0.000} C_DIS
LIN {X -84.292,Y -15.308,Z -16.884,A -90.000,B 90.000,C 0.000} C_DIS
LIN {X -83.915,Y -15.308,Z -16.529,A -90.000,B 90.000,C 0.000} C_DIS
LIN {X -83.561,Y -15.308,Z -16.266,A -90.000,B 90.000,C 0.000} C_DIS
LIN {X -83.213,Y -15.308,Z -16.046,A -90.000,B 90.000,C 0.000} C_DIS
LIN {X -82.832,Y -15.308,Z -15.825,A -90.000,B 90.000,C 0.000} C_DIS
LIN {X -82.429,Y -15.308,Z -15.634,A -90.000,B 90.000,C 0.000} C_DIS
LIN {X -81.980,Y -15.308,Z -15.447,A -90.000,B 90.000,C 0.000} C_DIS
LIN {X -81.552,Y -15.308,Z -15.291,A -90.000,B 90.000,C 0.000} C_DIS
LIN {X -80.966,Y -15.308,Z -15.137,A -90.000,B 90.000,C 0.000} C_DIS
LIN {X -80.523,Y -15.308,Z -15.028,A -90.000,B 90.000,C 0.000} C_DIS
LIN {X -79.384,Y -15.308,Z -14.873,A -90.000,B 90.000,C 0.000} C_DIS
LIN {X -79.068,Y -15.308,Z -14.846,A -90.000,B 90.000,C 0.000} C_DIS
LIN {X -78.051,Y -15.308,Z -14.824,A -90.000,B 90.000,C 0.000} C_DIS
LIN {X -77.584,Y -15.308,Z -14.833,A -90.000,B 90.000,C 0.000} C_DIS
LIN {X -77.407,Y -15.308,Z -14.848,A -90.000,B 90.000,C 0.000} C_DIS
LIN {X -76.427,Y -15.308,Z -14.959,A -90.000,B 90.000,C 0.000} C_DIS
LIN {X -76.054,Y -15.308,Z -15.016,A -90.000,B 90.000,C 0.000} C_DIS
LIN {X -74.960,Y -15.308,Z -15.274,A -90.000,B 90.000,C 0.000} C_DIS
LIN {X -74.797,Y -15.308,Z -15.316,A -90.000,B 90.000,C 0.000} C_DIS
LIN {X -74.553,Y -15.308,Z -15.380,A -90.000,B 90.000,C 0.000} C_DIS
LIN {X -74.330,Y -15.308,Z -15.447,A -90.000,B 90.000,C 0.000} C_DIS
LIN {X -73.890,Y -15.308,Z -15.602,A -90.000,B 90.000,C 0.000} C_DIS
LIN {X -72.739,Y -15.308,Z -16.034,A -90.000,B 90.000,C 0.000} C_DIS
LIN {X -72.473,Y -15.308,Z -16.137,A -90.000,B 90.000,C 0.000} C_DIS
LIN {X -71.791,Y -15.308,Z -16.462,A -90.000,B 90.000,C 0.000} C_DIS
LIN {X -70.707,Y -15.308,Z -17.001,A -90.000,B 90.000,C 0.000} C_DIS
LIN {X -69.533,Y -15.308,Z -17.658,A -90.000,B 90.000,C 0.000} C_DIS
LIN {X -69.106,Y -15.308,Z -17.891,A -90.000,B 90.000,C 0.000} C_DIS
LIN {X -68.207,Y -15.308,Z -18.414,A -90.000,B 90.000,C 0.000} C_DIS
LIN {X -67.072,Y -15.308,Z -19.079,A -90.000,B 90.000,C 0.000} C_DIS
LIN {X -66.345,Y -15.308,Z -19.534,A -90.000,B 90.000,C 0.000} C_DIS
LIN {X -66.059,Y -15.308,Z -19.723,A -90.000,B 90.000,C 0.000} C_DIS
LIN {X -65.041,Y -15.308,Z -20.411,A -90.000,B 90.000,C 0.000} C_DIS
LIN {X -64.613,Y -15.308,Z -20.709,A -90.000,B 90.000,C 0.000} C_DIS
LIN {X -64.572,Y -15.308,Z -20.742,A -90.000,B 90.000,C 0.000} C_DIS
LIN {X -63.589,Y -15.308,Z -21.456,A -90.000,B 90.000,C 0.000} C_DIS
LIN {X -62.811,Y -15.308,Z -22.038,A -90.000,B 90.000,C 0.000} C_DIS
LIN {X -62.536,Y -15.308,Z -22.263,A -90.000,B 90.000,C 0.000} C_DIS
LIN {X -62.182,Y -15.308,Z -22.520,A -90.000,B 90.000,C 0.000} C_DIS
LIN {X -61.575,Y -15.308,Z -22.971,A -90.000,B 90.000,C 0.000} C_DIS
LIN {X -60.934,Y -15.308,Z -23.405,A -90.000,B 90.000,C 0.000} C_DIS
LIN {X -60.137,Y -15.308,Z -23.850,A -90.000,B 90.000,C 0.000} C_DIS
LIN {X -59.139,Y -15.308,Z -24.299,A -90.000,B 90.000,C 0.000} C_DIS
LIN {X -58.886,Y -15.308,Z -24.390,A -90.000,B 90.000,C 0.000} C_DIS
LIN {X -57.746,Y -15.308,Z -24.809,A -90.000,B 90.000,C 0.000} C_DIS
LIN {X -56.911,Y -15.308,Z -25.072,A -90.000,B 90.000,C 0.000} C_DIS
LIN {X -56.153,Y -15.308,Z -25.302,A -90.000,B 90.000,C 0.000} C_DIS
LIN {X -55.418,Y -15.308,Z -25.502,A -90.000,B 90.000,C 0.000} C_DIS
LIN {X -53.928,Y -15.308,Z -25.881,A -90.000,B 90.000,C 0.000} C_DIS
LIN {X -53.758,Y -15.308,Z -25.921,A -90.000,B 90.000,C 0.000} C_DIS
LIN {X -53.358,Y -15.308,Z -26.004,A -90.000,B 90.000,C 0.000} C_DIS
LIN {X -52.074,Y -15.308,Z -26.294,A -90.000,B 90.000,C 0.000} C_DIS
LIN {X -51.460,Y -15.308,Z -26.418,A -90.000,B 90.000,C 0.000} C_DIS
LIN {X -50.720,Y -15.308,Z -26.552,A -90.000,B 90.000,C 0.000} C_DIS
LIN {X -49.148,Y -15.308,Z -26.801,A -90.000,B 90.000,C 0.000} C_DIS
LIN {X -48.925,Y -15.308,Z -26.839,A -90.000,B 90.000,C 0.000} C_DIS
LIN {X -48.688,Y -15.308,Z -26.878,A -90.000,B 90.000,C 0.000} C_DIS
LIN {X -47.274,Y -15.308,Z -27.070,A -90.000,B 90.000,C 0.000} C_DIS
LIN {X -45.681,Y -15.308,Z -27.288,A -90.000,B 90.000,C 0.000} C_DIS
LIN {X -45.468,Y -15.308,Z -27.320,A -90.000,B 90.000,C 0.000} C_DIS
LIN {X -45.134,Y -15.308,Z -27.374,A -90.000,B 90.000,C 0.000} C_DIS
LIN {X -42.644,Y -15.308,Z -27.744,A -90.000,B 90.000,C 0.000} C_DIS
LIN {X -41.240,Y -15.308,Z -27.985,A -90.000,B 90.000,C 0.000} C_DIS
LIN {X -40.765,Y -15.308,Z -28.059,A -90.000,B 90.000,C 0.000} C_DIS
LIN {X -40.211,Y -15.308,Z -28.158,A -90.000,B 90.000,C 0.000} C_DIS
LIN {X -38.948,Y -15.308,Z -28.403,A -90.000,B 90.000,C 0.000} C_DIS
LIN {X -38.111,Y -15.308,Z -28.569,A -90.000,B 90.000,C 0.000} C_DIS
LIN {X -37.631,Y -15.308,Z -28.674,A -90.000,B 90.000,C 0.000} C_DIS
LIN {X -36.287,Y -15.308,Z -28.949,A -90.000,B 90.000,C 0.000} C_DIS
LIN {X -35.880,Y -15.308,Z -29.038,A -90.000,B 90.000,C 0.000} C_DIS
LIN {X -33.668,Y -15.308,Z -29.533,A -90.000,B 90.000,C 0.000} C_DIS
LIN {X -31.924,Y -15.308,Z -29.927,A -90.000,B 90.000,C 0.000} C_DIS
LIN {X -31.366,Y -15.308,Z -30.057,A -90.000,B 90.000,C 0.000} C_DIS
LIN {X -29.124,Y -15.308,Z -30.554,A -90.000,B 90.000,C 0.000} C_DIS
LIN {X -28.322,Y -15.308,Z -30.710,A -90.000,B 90.000,C 0.000} C_DIS
LIN {X -27.054,Y -15.308,Z -30.941,A -90.000,B 90.000,C 0.000} C_DIS
LIN {X -26.891,Y -15.308,Z -30.968,A -90.000,B 90.000,C 0.000} C_DIS
LIN {X -26.277,Y -15.308,Z -31.047,A -90.000,B 90.000,C 0.000} C_DIS
LIN {X -25.589,Y -15.308,Z -31.107,A -90.000,B 90.000,C 0.000} C_DIS
LIN {X -25.195,Y -15.308,Z -31.117,A -90.000,B 90.000,C 0.000} C_DIS
LIN {X -24.833,Y -15.308,Z -31.134,A -90.000,B 90.000,C 0.000} C_DIS
LIN {X -24.722,Y -15.308,Z -31.129,A -90.000,B 90.000,C 0.000} C_DIS
LIN {X -24.089,Y -15.308,Z -31.119,A -90.000,B 90.000,C 0.000} C_DIS
LIN {X -23.457,Y -15.308,Z -31.131,A -90.000,B 90.000,C 0.000} C_DIS
LIN {X -22.916,Y -15.308,Z -31.135,A -90.000,B 90.000,C 0.000} C_DIS
LIN {X -22.298,Y -15.308,Z -31.167,A -90.000,B 90.000,C 0.000} C_DIS
LIN {X -21.608,Y -15.308,Z -31.208,A -90.000,B 90.000,C 0.000} C_DIS
LIN {X -21.257,Y -15.308,Z -31.235,A -90.000,B 90.000,C 0.000} C_DIS
LIN {X -19.802,Y -15.308,Z -31.381,A -90.000,B 90.000,C 0.000} C_DIS
LIN {X -19.160,Y -15.308,Z -31.449,A -90.000,B 90.000,C 0.000} C_DIS
LIN {X -18.248,Y -15.308,Z -31.559,A -90.000,B 90.000,C 0.000} C_DIS
LIN {X -16.625,Y -15.308,Z -31.787,A -90.000,B 90.000,C 0.000} C_DIS
LIN {X -15.389,Y -15.308,Z -32.006,A -90.000,B 90.000,C 0.000} C_DIS
LIN {X -15.216,Y -15.308,Z -32.039,A -90.000,B 90.000,C 0.000} C_DIS
LIN {X -13.626,Y -15.308,Z -32.358,A -90.000,B 90.000,C 0.000} C_DIS
LIN {X -12.657,Y -15.308,Z -32.526,A -90.000,B 90.000,C 0.000} C_DIS
LIN {X -12.284,Y -15.308,Z -32.596,A -90.000,B 90.000,C 0.000} C_DIS
LIN {X -11.902,Y -15.308,Z -32.674,A -90.000,B 90.000,C 0.000} C_DIS
LIN {X -10.755,Y -15.308,Z -32.859,A -90.000,B 90.000,C 0.000} C_DIS
LIN {X -9.520,Y -15.308,Z -33.084,A -90.000,B 90.000,C 0.000} C_DIS
LIN {X -8.420,Y -15.308,Z -33.282,A -90.000,B 90.000,C 0.000} C_DIS
LIN {X -6.917,Y -15.308,Z -33.588,A -90.000,B 90.000,C 0.000} C_DIS
LIN {X -6.384,Y -15.308,Z -33.677,A -90.000,B 90.000,C 0.000} C_DIS
LIN {X -4.735,Y -15.308,Z -33.982,A -90.000,B 90.000,C 0.000} C_DIS
LIN {X -3.756,Y -15.308,Z -34.127,A -90.000,B 90.000,C 0.000} C_DIS
LIN {X -1.023,Y -15.308,Z -34.499,A -90.000,B 90.000,C 0.000} C_DIS
LIN {X 0.037,Y -15.308,Z -34.639,A -90.000,B 90.000,C 0.000} C_DIS
LIN {X 0.201,Y -15.308,Z -34.663,A -90.000,B 90.000,C 0.000} C_DIS
LIN {X 0.436,Y -15.308,Z -34.697,A -90.000,B 90.000,C 0.000} C_DIS
LIN {X 1.942,Y -15.308,Z -34.939,A -90.000,B 90.000,C 0.000} C_DIS
LIN {X 2.849,Y -15.308,Z -35.091,A -90.000,B 90.000,C 0.000} C_DIS
LIN {X 4.246,Y -15.308,Z -35.334,A -90.000,B 90.000,C 0.000} C_DIS
LIN {X 4.524,Y -15.308,Z -35.377,A -90.000,B 90.000,C 0.000} C_DIS
LIN {X 6.442,Y -15.308,Z -35.737,A -90.000,B 90.000,C 0.000} C_DIS
LIN {X 7.197,Y -15.308,Z -35.872,A -90.000,B 90.000,C 0.000} C_DIS
LIN {X 7.275,Y -15.308,Z -35.886,A -90.000,B 90.000,C 0.000} C_DIS
LIN {X 8.659,Y -15.308,Z -36.190,A -90.000,B 90.000,C 0.000} C_DIS
LIN {X 9.726,Y -15.308,Z -36.421,A -90.000,B 90.000,C 0.000} C_DIS
LIN {X 11.058,Y -15.308,Z -36.736,A -90.000,B 90.000,C 0.000} C_DIS
LIN {X 13.389,Y -15.308,Z -37.256,A -90.000,B 90.000,C 0.000} C_DIS
LIN {X 14.285,Y -15.308,Z -37.439,A -90.000,B 90.000,C 0.000} C_DIS
LIN {X 15.541,Y -15.308,Z -37.653,A -90.000,B 90.000,C 0.000} C_DIS
LIN {X 16.407,Y -15.308,Z -37.780,A -90.000,B 90.000,C 0.000} C_DIS
LIN {X 17.210,Y -15.308,Z -37.821,A -90.000,B 90.000,C 0.000} C_DIS
LIN {X 17.857,Y -15.308,Z -37.805,A -90.000,B 90.000,C 0.000} C_DIS
LIN {X 18.231,Y -15.308,Z -37.789,A -90.000,B 90.000,C 0.000} C_DIS
LIN {X 18.899,Y -15.308,Z -37.715,A -90.000,B 90.000,C 0.000} C_DIS
LIN {X 19.765,Y -15.308,Z -37.643,A -90.000,B 90.000,C 0.000} C_DIS
LIN {X 21.293,Y -15.308,Z -37.470,A -90.000,B 90.000,C 0.000} C_DIS
LIN {X 21.535,Y -15.308,Z -37.445,A -90.000,B 90.000,C 0.000} C_DIS
LIN {X 21.983,Y -15.308,Z -37.402,A -90.000,B 90.000,C 0.000} C_DIS
LIN {X 22.853,Y -15.308,Z -37.337,A -90.000,B 90.000,C 0.000} C_DIS
LIN {X 23.566,Y -15.308,Z -37.306,A -90.000,B 90.000,C 0.000} C_DIS
LIN {X 24.493,Y -15.308,Z -37.259,A -90.000,B 90.000,C 0.000} C_DIS
LIN {X 26.007,Y -15.308,Z -37.204,A -90.000,B 90.000,C 0.000} C_DIS
LIN {X 26.430,Y -15.308,Z -37.194,A -90.000,B 90.000,C 0.000} C_DIS
LIN {X 26.598,Y -15.308,Z -37.195,A -90.000,B 90.000,C 0.000} C_DIS
LIN {X 27.576,Y -15.308,Z -37.176,A -90.000,B 90.000,C 0.000} C_DIS
LIN {X 28.080,Y -15.308,Z -37.186,A -90.000,B 90.000,C 0.000} C_DIS
LIN {X 28.229,Y -15.308,Z -37.191,A -90.000,B 90.000,C 0.000} C_DIS
LIN {X 29.108,Y -15.308,Z -37.196,A -90.000,B 90.000,C 0.000} C_DIS
LIN {X 30.065,Y -15.308,Z -37.211,A -90.000,B 90.000,C 0.000} C_DIS
LIN {X 31.171,Y -15.308,Z -37.248,A -90.000,B 90.000,C 0.000} C_DIS
LIN {X 32.167,Y -15.308,Z -37.260,A -90.000,B 90.000,C 0.000} C_DIS
LIN {X 32.974,Y -15.308,Z -37.286,A -90.000,B 90.000,C 0.000} C_DIS
LIN {X 34.402,Y -15.308,Z -37.348,A -90.000,B 90.000,C 0.000} C_DIS
LIN {X 34.595,Y -15.308,Z -37.364,A -90.000,B 90.000,C 0.000} C_DIS
LIN {X 35.803,Y -15.308,Z -37.434,A -90.000,B 90.000,C 0.000} C_DIS
LIN {X 37.254,Y -15.308,Z -37.577,A -90.000,B 90.000,C 0.000} C_DIS
LIN {X 38.538,Y -15.308,Z -37.763,A -90.000,B 90.000,C 0.000} C_DIS
LIN {X 40.061,Y -15.308,Z -38.010,A -90.000,B 90.000,C 0.000} C_DIS
LIN {X 40.515,Y -15.308,Z -38.095,A -90.000,B 90.000,C 0.000} C_DIS
LIN {X 43.140,Y -15.308,Z -38.735,A -90.000,B 90.000,C 0.000} C_DIS
LIN {X 43.358,Y -15.308,Z -38.786,A -90.000,B 90.000,C 0.000} C_DIS
LIN {X 43.876,Y -15.308,Z -38.939,A -90.000,B 90.000,C 0.000} C_DIS
LIN {X 45.212,Y -15.308,Z -39.382,A -90.000,B 90.000,C 0.000} C_DIS
LIN {X 46.625,Y -15.308,Z -39.879,A -90.000,B 90.000,C 0.000} C_DIS
LIN {X 47.100,Y -15.308,Z -40.077,A -90.000,B 90.000,C 0.000} C_DIS
LIN {X 47.144,Y -15.308,Z -40.096,A -90.000,B 90.000,C 0.000} C_DIS
LIN {X 49.495,Y -15.308,Z -41.119,A -90.000,B 90.000,C 0.000} C_DIS
LIN {X 49.741,Y -15.308,Z -41.245,A -90.000,B 90.000,C 0.000} C_DIS
LIN {X 52.187,Y -15.308,Z -42.544,A -90.000,B 90.000,C 0.000} C_DIS
LIN {X 52.552,Y -15.308,Z -42.742,A -90.000,B 90.000,C 0.000} C_DIS
LIN {X 52.702,Y -15.308,Z -42.825,A -90.000,B 90.000,C 0.000} C_DIS
LIN {X 55.114,Y -15.308,Z -44.347,A -90.000,B 90.000,C 0.000} C_DIS
LIN {X 55.508,Y -15.308,Z -44.614,A -90.000,B 90.000,C 0.000} C_DIS
LIN {X 57.720,Y -15.308,Z -46.256,A -90.000,B 90.000,C 0.000} C_DIS
LIN {X 60.122,Y -15.308,Z -48.286,A -90.000,B 90.000,C 0.000} C_DIS
LIN {X 61.033,Y -15.308,Z -49.006,A -90.000,B 90.000,C 0.000} C_DIS
LIN {X 61.707,Y -15.308,Z -49.496,A -90.000,B 90.000,C 0.000} C_DIS
LIN {X 62.531,Y -15.308,Z -50.051,A -90.000,B 90.000,C 0.000} C_DIS
LIN {X 63.424,Y -15.308,Z -50.613,A -90.000,B 90.000,C 0.000} C_DIS
LIN {X 64.665,Y -15.308,Z -51.333,A -90.000,B 90.000,C 0.000} C_DIS
LIN {X 65.327,Y -15.308,Z -51.724,A -90.000,B 90.000,C 0.000} C_DIS
LIN {X 66.933,Y -15.308,Z -52.606,A -90.000,B 90.000,C 0.000} C_DIS
LIN {X 67.843,Y -15.308,Z -53.096,A -90.000,B 90.000,C 0.000} C_DIS
LIN {X 70.123,Y -15.308,Z -54.376,A -90.000,B 90.000,C 0.000} C_DIS
LIN {X 72.320,Y -15.308,Z -55.694,A -90.000,B 90.000,C 0.000} C_DIS
LIN {X 74.549,Y -15.308,Z -57.161,A -90.000,B 90.000,C 0.000} C_DIS
LIN {X 74.768,Y -15.308,Z -57.307,A -90.000,B 90.000,C 0.000} C_DIS
LIN {X 75.927,Y -15.308,Z -58.163,A -90.000,B 90.000,C 0.000} C_DIS
LIN {X 76.545,Y -15.308,Z -58.627,A -90.000,B 90.000,C 0.000} C_DIS
LIN {X 77.309,Y -15.308,Z -59.260,A -90.000,B 90.000,C 0.000} C_DIS
LIN {X 78.146,Y -15.308,Z -59.957,A -90.000,B 90.000,C 0.000} C_DIS
LIN {X 78.183,Y -15.308,Z -59.988,A -90.000,B 90.000,C 0.000} C_DIS
LIN {X 78.502,Y -15.325,Z -60.261,A -90.000,B 90.000,C 0.000} C_DIS
LIN {X 78.789,Y -15.308,Z -60.504,A -90.000,B 90.000,C 0.000} C_DIS
LIN {X 78.973,Y -15.308,Z -60.657,A -90.000,B 90.000,C 0.000} C_DIS
LIN {X 78.977,Y -17.295,Z -60.660,A -90.000,B 90.000,C 0.000} C_DIS
LIN {X 78.985,Y -17.529,Z -60.667,A -90.000,B 90.000,C 0.000} C_DIS
LIN {X 79.016,Y -18.173,Z -60.692,A -90.000,B 90.000,C 0.000} C_DIS
LIN {X 79.046,Y -18.297,Z -60.718,A -90.000,B 90.000,C 0.000} C_DIS
LIN {X 79.164,Y -18.663,Z -60.814,A -90.000,B 90.000,C 0.000} C_DIS
LIN {X 79.275,Y -18.924,Z -60.902,A -90.000,B 90.000,C 0.000} C_DIS
LIN {X 79.379,Y -19.130,Z -60.984,A -90.000,B 90.000,C 0.000} C_DIS
LIN {X 79.477,Y -19.300,Z -61.059,A -90.000,B 90.000,C 0.000} C_DIS
LIN {X 79.569,Y -19.438,Z -61.127,A -90.000,B 90.000,C 0.000} C_DIS
LIN {X 79.655,Y -19.549,Z -61.188,A -90.000,B 90.000,C 0.000} C_DIS
LIN {X 79.735,Y -19.652,Z -61.243,A -90.000,B 90.000,C 0.000} C_DIS
LIN {X 79.809,Y -19.729,Z -61.290,A -90.000,B 90.000,C 0.000} C_DIS
LIN {X 79.827,Y -25.485,Z -61.301,A -90.000,B 90.000,C 0.000} C_DIS
LIN {X 79.829,Y -25.609,Z -61.302,A -90.000,B 90.000,C 0.000} C_DIS
LIN {X 79.836,Y -25.761,Z -61.306,A -90.000,B 90.000,C 0.000} C_DIS
LIN {X 79.844,Y -26.264,Z -61.312,A -90.000,B 90.000,C 0.000} C_DIS
LIN {X 79.878,Y -26.656,Z -61.331,A -90.000,B 90.000,C 0.000} C_DIS
LIN {X 79.942,Y -27.049,Z -61.366,A -90.000,B 90.000,C 0.000} C_DIS
LIN {X 80.002,Y -27.304,Z -61.394,A -90.000,B 90.000,C 0.000} C_DIS
LIN {X 80.056,Y -27.494,Z -61.415,A -90.000,B 90.000,C 0.000} C_DIS
LIN {X 80.107,Y -27.644,Z -61.430,A -90.000,B 90.000,C 0.000} C_DIS
LIN {X 80.153,Y -27.764,Z -61.439,A -90.000,B 90.000,C 0.000} C_DIS
LIN {X 80.195,Y -27.863,Z -61.442,A -90.000,B 90.000,C 0.000} C_DIS
LIN {X 80.234,Y -27.943,Z -61.438,A -90.000,B 90.000,C 0.000} C_DIS
LIN {X 80.269,Y -28.008,Z -61.428,A -90.000,B 90.000,C 0.000} C_DIS
LIN {X 80.301,Y -28.061,Z -61.413,A -90.000,B 90.000,C 0.000} C_DIS
LIN {X 80.329,Y -28.101,Z -61.391,A -90.000,B 90.000,C 0.000} C_DIS
LIN {X 80.355,Y -28.132,Z -61.363,A -90.000,B 90.000,C 0.000} C_DIS
LIN {X 80.367,Y -28.144,Z -61.348,A -90.000,B 90.000,C 0.000} C_DIS
LIN {X 80.390,Y -28.162,Z -61.311,A -90.000,B 90.000,C 0.000} C_DIS
LIN {X 80.400,Y -28.168,Z -61.291,A -90.000,B 90.000,C 0.000} C_DIS
LIN {X 80.419,Y -28.173,Z -61.246,A -90.000,B 90.000,C 0.000} C_DIS
LIN {X 80.436,Y -28.172,Z -61.196,A -90.000,B 90.000,C 0.000} C_DIS
LIN {X 80.451,Y -28.163,Z -61.140,A -90.000,B 90.000,C 0.000} C_DIS
LIN {X 80.465,Y -28.149,Z -61.079,A -90.000,B 90.000,C 0.000} C_DIS
LIN {X 80.478,Y -28.128,Z -61.012,A -90.000,B 90.000,C 0.000} C_DIS
LIN {X 80.501,Y -28.068,Z -60.862,A -90.000,B 90.000,C 0.000} C_DIS
LIN {X 80.511,Y -28.030,Z -60.780,A -90.000,B 90.000,C 0.000} C_DIS
LIN {X 80.531,Y -27.936,Z -60.599,A -90.000,B 90.000,C 0.000} C_DIS
LIN {X 80.552,Y -27.820,Z -60.399,A -90.000,B 90.000,C 0.000} C_DIS
LIN {X 80.575,Y -27.680,Z -60.179,A -90.000,B 90.000,C 0.000} C_DIS
LIN {X 80.602,Y -27.514,Z -59.940,A -90.000,B 90.000,C 0.000} C_DIS
LIN {X 80.618,Y -27.419,Z -59.813,A -90.000,B 90.000,C 0.000} C_DIS
LIN {X 80.635,Y -27.309,Z -59.683,A -90.000,B 90.000,C 0.000} C_DIS
LIN {X 80.676,Y -27.067,Z -59.408,A -90.000,B 90.000,C 0.000} C_DIS
LIN {X 80.700,Y -26.981,Z -59.264,A -90.000,B 90.000,C 0.000} C_DIS
LIN {X 80.726,Y -26.898,Z -59.115,A -90.000,B 90.000,C 0.000} C_DIS
LIN {X 80.788,Y -26.726,Z -58.806,A -90.000,B 90.000,C 0.000} C_DIS
LIN {X 80.863,Y -26.549,Z -58.481,A -90.000,B 90.000,C 0.000} C_DIS
LIN {X 80.906,Y -26.462,Z -58.313,A -90.000,B 90.000,C 0.000} C_DIS
LIN {X 80.953,Y -26.377,Z -58.141,A -90.000,B 90.000,C 0.000} C_DIS
LIN {X 81.004,Y -26.298,Z -57.965,A -90.000,B 90.000,C 0.000} C_DIS
LIN {X 81.060,Y -26.230,Z -57.785,A -90.000,B 90.000,C 0.000} C_DIS
LIN {X 81.120,Y -26.179,Z -57.602,A -90.000,B 90.000,C 0.000} C_DIS
LIN {X 81.185,Y -26.155,Z -57.415,A -90.000,B 90.000,C 0.000} C_DIS
LIN {X 81.256,Y -26.116,Z -57.224,A -90.000,B 90.000,C 0.000} C_DIS
LIN {X 81.293,Y -26.073,Z -57.128,A -90.000,B 90.000,C 0.000} C_DIS
LIN {X 81.331,Y -26.023,Z -57.030,A -90.000,B 90.000,C 0.000} C_DIS
LIN {X 81.412,Y -25.938,Z -56.833,A -90.000,B 90.000,C 0.000} C_DIS
LIN {X 81.455,Y -25.913,Z -56.733,A -90.000,B 90.000,C 0.000} C_DIS
LIN {X 81.499,Y -15.308,Z -56.633,A -90.000,B 90.000,C 0.000} C_DIS
LIN {X 81.700,Y -15.308,Z -56.182,A -90.000,B 90.000,C 0.000} C_DIS
LIN {X 82.134,Y -15.308,Z -55.110,A -90.000,B 90.000,C 0.000} C_DIS
LIN {X 82.335,Y -15.308,Z -54.666,A -90.000,B 90.000,C 0.000} C_DIS
LIN {X 83.331,Y -15.308,Z -52.811,A -90.000,B 90.000,C 0.000} C_DIS
LIN {X 83.577,Y -15.308,Z -52.389,A -90.000,B 90.000,C 0.000} C_DIS
LIN {X 84.758,Y -15.308,Z -50.656,A -90.000,B 90.000,C 0.000} C_DIS
LIN {X 85.025,Y -15.308,Z -50.291,A -90.000,B 90.000,C 0.000} C_DIS
LIN {X 86.337,Y -15.308,Z -48.714,A -90.000,B 90.000,C 0.000} C_DIS
LIN {X 86.664,Y -15.308,Z -48.352,A -90.000,B 90.000,C 0.000} C_DIS
LIN {X 88.117,Y -15.308,Z -46.880,A -90.000,B 90.000,C 0.000} C_DIS
LIN {X 88.479,Y -15.308,Z -46.553,A -90.000,B 90.000,C 0.000} C_DIS
LIN {X 90.061,Y -15.308,Z -45.164,A -90.000,B 90.000,C 0.000} C_DIS
LIN {X 91.751,Y -15.308,Z -43.851,A -90.000,B 90.000,C 0.000} C_DIS
LIN {X 92.110,Y -15.308,Z -43.588,A -90.000,B 90.000,C 0.000} C_DIS
LIN {X 93.780,Y -15.308,Z -42.419,A -90.000,B 90.000,C 0.000} C_DIS
LIN {X 95.417,Y -15.308,Z -41.383,A -90.000,B 90.000,C 0.000} C_DIS
LIN {X 95.838,Y -15.308,Z -41.136,A -90.000,B 90.000,C 0.000} C_DIS
LIN {X 97.376,Y -15.308,Z -40.260,A -90.000,B 90.000,C 0.000} C_DIS
LIN {X 98.805,Y -15.308,Z -39.523,A -90.000,B 90.000,C 0.000} C_DIS
LIN {X 98.814,Y -15.308,Z -39.518,A -90.000,B 90.000,C 0.000} C_DIS
LIN {X 98.814,Y -60.000,Z -39.518,A -90.000,B 90.000,C 0.000} C_DIS
LIN {X 105.145,Y -60.000,Z -77.014,A -90.000,B 90.000,C 0.000} C_DIS
LIN {X 105.145,Y -15.308,Z -77.014,A -90.000,B 90.000,C 0.000} C_DIS
LIN {X 104.209,Y -15.308,Z -78.763,A -90.000,B 90.000,C 0.000} C_DIS
LIN {X 103.987,Y -15.308,Z -79.149,A -90.000,B 90.000,C 0.000} C_DIS
LIN {X 103.058,Y -15.308,Z -80.726,A -90.000,B 90.000,C 0.000} C_DIS
LIN {X 102.198,Y -15.308,Z -82.078,A -90.000,B 90.000,C 0.000} C_DIS
LIN {X 99.737,Y -15.308,Z -85.762,A -90.000,B 90.000,C 0.000} C_DIS
LIN {X 99.868,Y -15.308,Z -87.446,A -90.000,B 90.000,C 0.000} C_DIS
LIN {X 100.035,Y -15.308,Z -89.825,A -90.000,B 90.000,C 0.000} C_DIS
LIN {X 100.315,Y -15.308,Z -90.386,A -90.000,B 90.000,C 0.000} C_DIS
LIN {X 100.428,Y -15.308,Z -90.672,A -90.000,B 90.000,C 0.000} C_DIS
LIN {X 100.788,Y -15.308,Z -91.512,A -90.000,B 90.000,C 0.000} C_DIS
LIN {X 100.840,Y -15.308,Z -91.629,A -90.000,B 90.000,C 0.000} C_DIS
LIN {X 100.998,Y -15.308,Z -92.044,A -90.000,B 90.000,C 0.000} C_DIS
LIN {X 101.066,Y -15.308,Z -92.232,A -90.000,B 90.000,C 0.000} C_DIS
LIN {X 101.387,Y -15.308,Z -93.200,A -90.000,B 90.000,C 0.000} C_DIS
LIN {X 101.556,Y -15.308,Z -93.805,A -90.000,B 90.000,C 0.000} C_DIS
LIN {X 101.654,Y -15.308,Z -94.168,A -90.000,B 90.000,C 0.000} C_DIS
LIN {X 101.818,Y -15.308,Z -94.828,A -90.000,B 90.000,C 0.000} C_DIS
LIN {X 101.903,Y -15.308,Z -95.188,A -90.000,B 90.000,C 0.000} C_DIS
LIN {X 102.044,Y -15.308,Z -95.906,A -90.000,B 90.000,C 0.000} C_DIS
LIN {X 102.109,Y -15.308,Z -96.216,A -90.000,B 90.000,C 0.000} C_DIS
LIN {X 102.237,Y -15.308,Z -96.957,A -90.000,B 90.000,C 0.000} C_DIS
LIN {X 102.313,Y -15.308,Z -97.317,A -90.000,B 90.000,C 0.000} C_DIS
LIN {X 102.466,Y -15.308,Z -98.160,A -90.000,B 90.000,C 0.000} C_DIS
LIN {X 102.612,Y -15.308,Z -98.858,A -90.000,B 90.000,C 0.000} C_DIS
LIN {X 102.731,Y -15.308,Z -99.513,A -90.000,B 90.000,C 0.000} C_DIS
LIN {X 102.867,Y -15.308,Z -100.205,A -90.000,B 90.000,C 0.000} C_DIS
LIN {X 103.075,Y -15.308,Z -101.358,A -90.000,B 90.000,C 0.000} C_DIS
LIN {X 103.153,Y -15.308,Z -101.787,A -90.000,B 90.000,C 0.000} C_DIS
LIN {X 103.442,Y -15.308,Z -103.491,A -90.000,B 90.000,C 0.000} C_DIS
LIN {X 103.812,Y -15.308,Z -105.803,A -90.000,B 90.000,C 0.000} C_DIS
LIN {X 104.129,Y -15.308,Z -107.872,A -90.000,B 90.000,C 0.000} C_DIS
LIN {X 104.197,Y -15.308,Z -108.329,A -90.000,B 90.000,C 0.000} C_DIS
LIN {X 104.436,Y -15.308,Z -110.036,A -90.000,B 90.000,C 0.000} C_DIS
LIN {X 104.565,Y -15.308,Z -110.978,A -90.000,B 90.000,C 0.000} C_DIS
LIN {X 104.729,Y -15.308,Z -112.302,A -90.000,B 90.000,C 0.000} C_DIS
LIN {X 104.894,Y -15.308,Z -113.650,A -90.000,B 90.000,C 0.000} C_DIS
LIN {X 105.170,Y -15.308,Z -116.309,A -90.000,B 90.000,C 0.000} C_DIS
LIN {X 105.407,Y -15.308,Z -119.030,A -90.000,B 90.000,C 0.000} C_DIS
LIN {X 105.553,Y -15.308,Z -120.978,A -90.000,B 90.000,C 0.000} C_DIS
LIN {X 105.601,Y -15.308,Z -121.543,A -90.000,B 90.000,C 0.000} C_DIS
LIN {X 105.687,Y -15.308,Z -122.810,A -90.000,B 90.000,C 0.000} C_DIS
LIN {X 105.781,Y -15.308,Z -124.082,A -90.000,B 90.000,C 0.000} C_DIS
LIN {X 105.873,Y -15.308,Z -125.551,A -90.000,B 90.000,C 0.000} C_DIS
LIN {X 105.937,Y -15.308,Z -126.628,A -90.000,B 90.000,C 0.000} C_DIS
LIN {X 105.958,Y -15.308,Z -127.031,A -90.000,B 90.000,C 0.000} C_DIS
LIN {X 106.073,Y -15.308,Z -129.555,A -90.000,B 90.000,C 0.000} C_DIS
LIN {X 106.137,Y -15.308,Z -132.139,A -90.000,B 90.000,C 0.000} C_DIS
LIN {X 106.139,Y -15.308,Z -132.229,A -90.000,B 90.000,C 0.000} C_DIS
LIN {X 106.145,Y -15.308,Z -134.413,A -90.000,B 90.000,C 0.000} C_DIS
LIN {X 106.149,Y -15.308,Z -135.192,A -90.000,B 90.000,C 0.000} C_DIS
LIN {X 106.119,Y -15.308,Z -137.216,A -90.000,B 90.000,C 0.000} C_DIS
LIN {X 106.095,Y -15.308,Z -138.520,A -90.000,B 90.000,C 0.000} C_DIS
LIN {X 106.033,Y -15.308,Z -140.543,A -90.000,B 90.000,C 0.000} C_DIS
LIN {X 105.969,Y -15.308,Z -142.380,A -90.000,B 90.000,C 0.000} C_DIS
LIN {X 105.864,Y -15.308,Z -144.628,A -90.000,B 90.000,C 0.000} C_DIS
LIN {X 105.788,Y -15.308,Z -146.159,A -90.000,B 90.000,C 0.000} C_DIS
LIN {X 105.545,Y -15.308,Z -150.015,A -90.000,B 90.000,C 0.000} C_DIS
LIN {X 105.401,Y -15.308,Z -151.853,A -90.000,B 90.000,C 0.000} C_DIS
LIN {X 105.239,Y -15.308,Z -153.857,A -90.000,B 90.000,C 0.000} C_DIS
LIN {X 105.077,Y -15.308,Z -155.660,A -90.000,B 90.000,C 0.000} C_DIS
LIN {X 104.873,Y -15.308,Z -157.814,A -90.000,B 90.000,C 0.000} C_DIS
LIN {X 104.574,Y -15.308,Z -160.839,A -90.000,B 90.000,C 0.000} C_DIS
LIN {X 104.197,Y -15.308,Z -164.441,A -90.000,B 90.000,C 0.000} C_DIS
LIN {X 104.095,Y -15.308,Z -165.364,A -90.000,B 90.000,C 0.000} C_DIS
LIN {X 103.814,Y -15.308,Z -167.975,A -90.000,B 90.000,C 0.000} C_DIS
LIN {X 103.716,Y -15.308,Z -168.841,A -90.000,B 90.000,C 0.000} C_DIS
LIN {X 103.431,Y -15.308,Z -171.386,A -90.000,B 90.000,C 0.000} C_DIS
LIN {X 103.048,Y -15.308,Z -174.619,A -90.000,B 90.000,C 0.000} C_DIS
LIN {X 102.958,Y -15.308,Z -175.333,A -90.000,B 90.000,C 0.000} C_DIS
LIN {X 102.663,Y -15.308,Z -177.627,A -90.000,B 90.000,C 0.000} C_DIS
LIN {X 102.581,Y -15.308,Z -178.242,A -90.000,B 90.000,C 0.000} C_DIS
LIN {X 102.450,Y -15.308,Z -179.143,A -90.000,B 90.000,C 0.000} C_DIS
LIN {X 102.115,Y -15.308,Z -181.482,A -90.000,B 90.000,C 0.000} C_DIS
LIN {X 101.733,Y -15.308,Z -183.966,A -90.000,B 90.000,C 0.000} C_DIS
LIN {X 100.952,Y -15.308,Z -188.887,A -90.000,B 90.000,C 0.000} C_DIS
LIN {X 100.556,Y -15.308,Z -191.514,A -90.000,B 90.000,C 0.000} C_DIS
LIN {X 100.135,Y -15.308,Z -194.235,A -90.000,B 90.000,C 0.000} C_DIS
LIN {X 99.963,Y -15.308,Z -195.322,A -90.000,B 90.000,C 0.000} C_DIS
LIN {X 99.638,Y -15.308,Z -197.280,A -90.000,B 90.000,C 0.000} C_DIS
LIN {X 99.424,Y -15.308,Z -198.555,A -90.000,B 90.000,C 0.000} C_DIS
LIN {X 98.694,Y -15.308,Z -202.630,A -90.000,B 90.000,C 0.000} C_DIS
LIN {X 98.229,Y -15.308,Z -205.026,A -90.000,B 90.000,C 0.000} C_DIS
LIN {X 97.771,Y -15.308,Z -207.423,A -90.000,B 90.000,C 0.000} C_DIS
LIN {X 97.521,Y -15.308,Z -208.663,A -90.000,B 90.000,C 0.000} C_DIS
LIN {X 96.415,Y -15.308,Z -214.028,A -90.000,B 90.000,C 0.000} C_DIS
LIN {X 96.211,Y -15.308,Z -214.956,A -90.000,B 90.000,C 0.000} C_DIS
LIN {X 95.165,Y -15.308,Z -219.604,A -90.000,B 90.000,C 0.000} C_DIS
LIN {X 94.944,Y -15.308,Z -220.540,A -90.000,B 90.000,C 0.000} C_DIS
LIN {X 94.851,Y -15.308,Z -220.925,A -90.000,B 90.000,C 0.000} C_DIS
LIN {X 94.643,Y -15.308,Z -221.746,A -90.000,B 90.000,C 0.000} C_DIS
LIN {X 93.466,Y -15.308,Z -226.467,A -90.000,B 90.000,C 0.000} C_DIS
LIN {X 91.906,Y -15.308,Z -232.132,A -90.000,B 90.000,C 0.000} C_DIS
LIN {X 90.132,Y -15.308,Z -238.013,A -90.000,B 90.000,C 0.000} C_DIS
LIN {X 89.809,Y -15.308,Z -238.993,A -90.000,B 90.000,C 0.000} C_DIS
LIN {X 88.317,Y -15.308,Z -243.561,A -90.000,B 90.000,C 0.000} C_DIS
LIN {X 88.317,Y -60.000,Z -243.561,A -90.000,B 90.000,C 0.000} C_DIS
LIN {X 99.925,Y -60.000,Z -88.260,A -90.000,B 90.000,C 0.000} C_DIS
LIN {X 99.925,Y -13.308,Z -88.260,A -90.000,B 90.000,C 0.000} C_DIS
LIN {X 100.078,Y -13.313,Z -88.521,A -90.000,B 90.000,C 0.000} C_DIS
LIN {X 100.165,Y -13.319,Z -88.690,A -90.000,B 90.000,C 0.000} C_DIS
LIN {X 100.263,Y -13.330,Z -88.882,A -90.000,B 90.000,C 0.000} C_DIS
LIN {X 100.351,Y -13.343,Z -89.058,A -90.000,B 90.000,C 0.000} C_DIS
LIN {X 100.523,Y -13.376,Z -89.410,A -90.000,B 90.000,C 0.000} C_DIS
LIN {X 100.642,Y -13.406,Z -89.659,A -90.000,B 90.000,C 0.000} C_DIS
LIN {X 100.908,Y -13.412,Z -90.163,A -90.000,B 90.000,C 0.000} C_DIS
LIN {X 101.027,Y -13.417,Z -90.421,A -90.000,B 90.000,C 0.000} C_DIS
LIN {X 101.459,Y -13.427,Z -91.348,A -90.000,B 90.000,C 0.000} C_DIS
LIN {X 101.661,Y -13.430,Z -91.857,A -90.000,B 90.000,C 0.000} C_DIS
LIN {X 102.060,Y -13.444,Z -92.930,A -90.000,B 90.000,C 0.000} C_DIS
LIN {X 102.198,Y -13.447,Z -93.383,A -90.000,B 90.000,C 0.000} C_DIS
LIN {X 102.394,Y -13.455,Z -94.031,A -90.000,B 90.000,C 0.000} C_DIS
LIN {X 102.517,Y -13.460,Z -94.476,A -90.000,B 90.000,C 0.000} C_DIS
LIN {X 102.613,Y -13.462,Z -94.854,A -90.000,B 90.000,C 0.000} C_DIS
LIN {X 102.679,Y -13.465,Z -95.116,A -90.000,B 90.000,C 0.000} C_DIS
LIN {X 102.753,Y -13.471,Z -95.418,A -90.000,B 90.000,C 0.000} C_DIS
LIN {X 102.907,Y -13.478,Z -96.106,A -90.000,B 90.000,C 0.000} C_DIS
LIN {X 102.979,Y -13.484,Z -96.444,A -90.000,B 90.000,C 0.000} C_DIS
LIN {X 103.066,Y -13.489,Z -96.865,A -90.000,B 90.000,C 0.000} C_DIS
LIN {X 103.138,Y -13.490,Z -97.203,A -90.000,B 90.000,C 0.000} C_DIS
LIN {X 103.304,Y -13.499,Z -98.005,A -90.000,B 90.000,C 0.000} C_DIS
LIN {X 103.464,Y -13.499,Z -98.784,A -90.000,B 90.000,C 0.000} C_DIS
LIN {X 103.578,Y -13.502,Z -99.359,A -90.000,B 90.000,C 0.000} C_DIS
LIN {X 103.703,Y -13.502,Z -100.007,A -90.000,B 90.000,C 0.000} C_DIS
LIN {X 103.876,Y -13.505,Z -100.927,A -90.000,B 90.000,C 0.000} C_DIS
LIN {X 104.034,Y -13.506,Z -101.808,A -90.000,B 90.000,C 0.000} C_DIS
LIN {X 104.216,Y -13.508,Z -102.847,A -90.000,B 90.000,C 0.000} C_DIS
LIN {X 104.365,Y -13.509,Z -103.734,A -90.000,B 90.000,C 0.000} C_DIS
LIN {X 104.671,Y -13.511,Z -105.615,A -90.000,B 90.000,C 0.000} C_DIS
LIN {X 105.046,Y -13.511,Z -108.077,A -90.000,B 90.000,C 0.000} C_DIS
LIN {X 105.386,Y -13.511,Z -110.514,A -90.000,B 90.000,C 0.000} C_DIS
LIN {X 105.511,Y -13.511,Z -111.477,A -90.000,B 90.000,C 0.000} C_DIS
LIN {X 105.715,Y -13.514,Z -113.080,A -90.000,B 90.000,C 0.000} C_DIS
LIN {X 105.771,Y -13.513,Z -113.559,A -90.000,B 90.000,C 0.000} C_DIS
LIN {X 105.957,Y -13.519,Z -115.243,A -90.000,B 90.000,C 0.000} C_DIS
LIN {X 106.057,Y -13.518,Z -116.231,A -90.000,B 90.000,C 0.000} C_DIS
LIN {X 106.183,Y -13.523,Z -117.563,A -90.000,B 90.000,C 0.000} C_DIS
LIN {X 106.297,Y -13.521,Z -118.898,A -90.000,B 90.000,C 0.000} C_DIS
LIN {X 106.389,Y -13.524,Z -120.044,A -90.000,B 90.000,C 0.000} C_DIS
LIN {X 106.459,Y -13.524,Z -120.985,A -90.000,B 90.000,C 0.000} C_DIS
LIN {X 106.497,Y -13.521,Z -121.502,A -90.000,B 90.000,C 0.000} C_DIS
LIN {X 106.585,Y -13.523,Z -122.743,A -90.000,B 90.000,C 0.000} C_DIS
LIN {X 106.630,Y -13.521,Z -123.393,A -90.000,B 90.000,C 0.000} C_DIS
LIN {X 106.681,Y -13.518,Z -124.210,A -90.000,B 90.000,C 0.000} C_DIS
LIN {X 106.756,Y -13.516,Z -125.471,A -90.000,B 90.000,C 0.000} C_DIS
LIN {X 106.835,Y -13.517,Z -126.784,A -90.000,B 90.000,C 0.000} C_DIS
LIN {X 106.848,Y -13.518,Z -127.021,A -90.000,B 90.000,C 0.000} C_DIS
LIN {X 106.907,Y -13.518,Z -128.300,A -90.000,B 90.000,C 0.000} C_DIS
LIN {X 106.969,Y -13.520,Z -129.575,A -90.000,B 90.000,C 0.000} C_DIS
LIN {X 107.019,Y -13.524,Z -131.297,A -90.000,B 90.000,C 0.000} C_DIS
LIN {X 107.050,Y -13.528,Z -132.261,A -90.000,B 90.000,C 0.000} C_DIS
LIN {X 107.069,Y -13.535,Z -134.012,A -90.000,B 90.000,C 0.000} C_DIS
LIN {X 107.086,Y -13.541,Z -135.174,A -90.000,B 90.000,C 0.000} C_DIS
LIN {X 107.082,Y -13.550,Z -136.503,A -90.000,B 90.000,C 0.000} C_DIS
LIN {X 107.072,Y -13.557,Z -137.930,A -90.000,B 90.000,C 0.000} C_DIS
LIN {X 107.067,Y -13.560,Z -138.490,A -90.000,B 90.000,C 0.000} C_DIS
LIN {X 107.045,Y -13.567,Z -139.638,A -90.000,B 90.000,C 0.000} C_DIS
LIN {X 106.987,Y -13.578,Z -141.983,A -90.000,B 90.000,C 0.000} C_DIS
LIN {X 106.977,Y -13.578,Z -142.278,A -90.000,B 90.000,C 0.000} C_DIS
LIN {X 106.881,Y -13.591,Z -144.807,A -90.000,B 90.000,C 0.000} C_DIS
LIN {X 106.844,Y -13.594,Z -145.675,A -90.000,B 90.000,C 0.000} C_DIS
LIN {X 106.816,Y -13.593,Z -146.203,A -90.000,B 90.000,C 0.000} C_DIS
LIN {X 106.682,Y -13.600,Z -148.499,A -90.000,B 90.000,C 0.000} C_DIS
LIN {X 106.616,Y -13.600,Z -149.563,A -90.000,B 90.000,C 0.000} C_DIS
LIN {X 106.577,Y -13.596,Z -150.074,A -90.000,B 90.000,C 0.000} C_DIS
LIN {X 106.279,Y -13.592,Z -153.737,A -90.000,B 90.000,C 0.000} C_DIS
LIN {X 106.084,Y -13.583,Z -155.755,A -90.000,B 90.000,C 0.000} C_DIS
LIN {X 105.882,Y -13.577,Z -157.791,A -90.000,B 90.000,C 0.000} C_DIS
LIN {X 105.538,Y -13.559,Z -160.940,A -90.000,B 90.000,C 0.000} C_DIS
LIN {X 105.459,Y -13.556,Z -161.639,A -90.000,B 90.000,C 0.000} C_DIS
LIN {X 105.119,Y -13.537,Z -164.545,A -90.000,B 90.000,C 0.000} C_DIS
LIN {X 104.991,Y -13.531,Z -165.623,A -90.000,B 90.000,C 0.000} C_DIS
LIN {X 104.736,Y -13.518,Z -167.737,A -90.000,B 90.000,C 0.000} C_DIS
LIN {X 104.693,Y -13.516,Z -168.094,A -90.000,B 90.000,C 0.000} C_DIS
LIN {X 104.581,Y -13.511,Z -169.012,A -90.000,B 90.000,C 0.000} C_DIS
LIN {X 104.384,Y -13.501,Z -170.572,A -90.000,B 90.000,C 0.000} C_DIS
LIN {X 104.174,Y -13.493,Z -172.253,A -90.000,B 90.000,C 0.000} C_DIS
LIN {X 103.894,Y -13.480,Z -174.368,A -90.000,B 90.000,C 0.000} C_DIS
LIN {X 103.741,Y -13.476,Z -175.530,A -90.000,B 90.000,C 0.000} C_DIS
LIN {X 103.433,Y -13.465,Z -177.731,A -90.000,B 90.000,C 0.000} C_DIS
LIN {X 103.305,Y -13.464,Z -178.636,A -90.000,B 90.000,C 0.000} C_DIS
LIN {X 103.185,Y -13.463,Z -179.449,A -90.000,B 90.000,C 0.000} C_DIS
LIN {X 102.855,Y -13.456,Z -181.626,A -90.000,B 90.000,C 0.000} C_DIS
LIN {X 102.447,Y -13.452,Z -184.220,A -90.000,B 90.000,C 0.000} C_DIS
LIN {X 101.795,Y -13.450,Z -188.294,A -90.000,B 90.000,C 0.000} C_DIS
LIN {X 101.605,Y -13.449,Z -189.493,A -90.000,B 90.000,C 0.000} C_DIS
LIN {X 101.412,Y -13.448,Z -190.757,A -90.000,B 90.000,C 0.000} C_DIS
LIN {X 101.308,Y -13.447,Z -191.430,A -90.000,B 90.000,C 0.000} C_DIS
LIN {X 101.224,Y -13.446,Z -191.959,A -90.000,B 90.000,C 0.000} C_DIS
LIN {X 100.939,Y -13.445,Z -193.806,A -90.000,B 90.000,C 0.000} C_DIS
LIN {X 100.798,Y -13.443,Z -194.666,A -90.000,B 90.000,C 0.000} C_DIS
LIN {X 100.668,Y -13.443,Z -195.487,A -90.000,B 90.000,C 0.000} C_DIS
LIN {X 100.472,Y -13.448,Z -196.739,A -90.000,B 90.000,C 0.000} C_DIS
LIN {X 100.149,Y -13.449,Z -198.686,A -90.000,B 90.000,C 0.000} C_DIS
LIN {X 99.879,Y -13.458,Z -200.314,A -90.000,B 90.000,C 0.000} C_DIS
LIN {X 99.451,Y -13.463,Z -202.777,A -90.000,B 90.000,C 0.000} C_DIS
LIN {X 99.117,Y -13.478,Z -204.675,A -90.000,B 90.000,C 0.000} C_DIS
LIN {X 98.543,Y -13.486,Z -207.766,A -90.000,B 90.000,C 0.000} C_DIS
LIN {X 98.187,Y -13.499,Z -209.660,A -90.000,B 90.000,C 0.000} C_DIS
LIN {X 98.114,Y -13.501,Z -210.029,A -90.000,B 90.000,C 0.000} C_DIS
LIN {X 97.272,Y -13.511,Z -214.217,A -90.000,B 90.000,C 0.000} C_DIS
LIN {X 97.030,Y -13.521,Z -215.399,A -90.000,B 90.000,C 0.000} C_DIS
LIN {X 95.992,Y -13.531,Z -220.094,A -90.000,B 90.000,C 0.000} C_DIS
LIN {X 95.807,Y -13.537,Z -220.917,A -90.000,B 90.000,C 0.000} C_DIS
LIN {X 94.488,Y -13.543,Z -226.251,A -90.000,B 90.000,C 0.000} C_DIS
LIN {X 94.415,Y -13.542,Z -226.543,A -90.000,B 90.000,C 0.000} C_DIS
LIN {X 94.369,Y -13.541,Z -226.716,A -90.000,B 90.000,C 0.000} C_DIS
LIN {X 93.156,Y -13.544,Z -231.140,A -90.000,B 90.000,C 0.000} C_DIS
LIN {X 92.859,Y -13.544,Z -232.223,A -90.000,B 90.000,C 0.000} C_DIS
LIN {X 92.806,Y -13.543,Z -232.403,A -90.000,B 90.000,C 0.000} C_DIS
LIN {X 91.594,Y -13.545,Z -236.435,A -90.000,B 90.000,C 0.000} C_DIS
LIN {X 91.064,Y -13.547,Z -238.202,A -90.000,B 90.000,C 0.000} C_DIS
LIN {X 90.969,Y -13.548,Z -238.507,A -90.000,B 90.000,C 0.000} C_DIS
LIN {X 89.327,Y -13.554,Z -243.561,A -90.000,B 90.000,C 0.000} C_DIS
LIN {X 89.327,Y -60.000,Z -243.561,A -90.000,B 90.000,C 0.000} C_DIS
LIN {X -119.190,Y -60.000,Z -243.561,A -90.000,B 90.000,C 0.000} C_DIS
LIN {X -119.190,Y -14.438,Z -243.561,A -90.000,B 90.000,C 0.000} C_DIS
LIN {X -119.102,Y -14.308,Z -243.308,A -90.000,B 90.000,C 0.000} C_DIS
LIN {X -119.058,Y -14.260,Z -243.221,A -90.000,B 90.000,C 0.000} C_DIS
LIN {X -118.859,Y -14.117,Z -242.914,A -90.000,B 90.000,C 0.000} C_DIS
LIN {X -118.842,Y -14.108,Z -242.893,A -90.000,B 90.000,C 0.000} C_DIS
LIN {X -118.723,Y -14.058,Z -242.751,A -90.000,B 90.000,C 0.000} C_DIS
LIN {X -118.625,Y -14.029,Z -242.648,A -90.000,B 90.000,C 0.000} C_DIS
LIN {X -118.404,Y -13.991,Z -242.450,A -90.000,B 90.000,C 0.000} C_DIS
LIN {X -118.258,Y -13.983,Z -242.342,A -90.000,B 90.000,C 0.000} C_DIS
LIN {X -116.426,Y -13.961,Z -241.060,A -90.000,B 90.000,C 0.000} C_DIS
LIN {X -115.827,Y -13.958,Z -240.640,A -90.000,B 90.000,C 0.000} C_DIS
LIN {X -114.799,Y -13.951,Z -239.929,A -90.000,B 90.000,C 0.000} C_DIS
LIN {X -110.276,Y -13.909,Z -236.797,A -90.000,B 90.000,C 0.000} C_DIS
LIN {X -108.503,Y -13.893,Z -235.571,A -90.000,B 90.000,C 0.000} C_DIS
LIN {X -104.937,Y -13.864,Z -233.138,A -90.000,B 90.000,C 0.000} C_DIS
LIN {X -100.883,Y -13.833,Z -230.374,A -90.000,B 90.000,C 0.000} C_DIS
LIN {X -99.660,Y -13.823,Z -229.553,A -90.000,B 90.000,C 0.000} C_DIS
LIN {X -94.931,Y -13.810,Z -226.407,A -90.000,B 90.000,C 0.000} C_DIS
LIN {X -92.997,Y -13.805,Z -225.118,A -90.000,B 90.000,C 0.000} C_DIS
LIN {X -92.033,Y -13.802,Z -224.488,A -90.000,B 90.000,C 0.000} C_DIS
LIN {X -85.574,Y -13.798,Z -220.283,A -90.000,B 90.000,C 0.000} C_DIS
LIN {X -84.896,Y -13.796,Z -219.844,A -90.000,B 90.000,C 0.000} C_DIS
LIN {X -84.706,Y -13.794,Z -219.722,A -90.000,B 90.000,C 0.000} C_DIS
LIN {X -78.307,Y -13.779,Z -215.658,A -90.000,B 90.000,C 0.000} C_DIS
LIN {X -76.650,Y -13.769,Z -214.616,A -90.000,B 90.000,C 0.000} C_DIS
LIN {X -70.671,Y -13.730,Z -210.888,A -90.000,B 90.000,C 0.000} C_DIS
LIN {X -68.274,Y -13.712,Z -209.399,A -90.000,B 90.000,C 0.000} C_DIS
LIN {X -66.831,Y -13.702,Z -208.498,A -90.000,B 90.000,C 0.000} C_DIS
LIN {X -62.948,Y -13.678,Z -206.076,A -90.000,B 90.000,C 0.000} C_DIS
LIN {X -61.658,Y -13.668,Z -205.275,A -90.000,B 90.000,C 0.000} C_DIS
LIN {X -60.486,Y -13.658,Z -204.547,A -90.000,B 90.000,C 0.000} C_DIS
LIN {X -56.869,Y -13.635,Z -202.257,A -90.000,B 90.000,C 0.000} C_DIS
LIN {X -53.875,Y -13.613,Z -200.381,A -90.000,B 90.000,C 0.000} C_DIS
LIN {X -51.874,Y -13.596,Z -199.081,A -90.000,B 90.000,C 0.000} C_DIS
LIN {X -50.163,Y -13.583,Z -197.968,A -90.000,B 90.000,C 0.000} C_DIS
LIN {X -48.485,Y -13.579,Z -196.872,A -90.000,B 90.000,C 0.000} C_DIS
LIN {X -48.314,Y -13.580,Z -196.758,A -90.000,B 90.000,C 0.000} C_DIS
LIN {X -44.712,Y -13.562,Z -194.330,A -90.000,B 90.000,C 0.000} C_DIS
LIN {X -43.807,Y -13.560,Z -193.713,A -90.000,B 90.000,C 0.000} C_DIS
LIN {X -41.849,Y -13.549,Z -192.336,A -90.000,B 90.000,C 0.000} C_DIS
LIN {X -40.262,Y -13.543,Z -191.223,A -90.000,B 90.000,C 0.000} C_DIS
LIN {X -39.798,Y -13.544,Z -190.892,A -90.000,B 90.000,C 0.000} C_DIS
LIN {X -36.608,Y -13.531,Z -188.565,A -90.000,B 90.000,C 0.000} C_DIS
LIN {X -36.355,Y -13.531,Z -188.378,A -90.000,B 90.000,C 0.000} C_DIS
LIN {X -34.874,Y -13.526,Z -187.268,A -90.000,B 90.000,C 0.000} C_DIS
LIN {X -33.265,Y -13.520,Z -186.065,A -90.000,B 90.000,C 0.000} C_DIS
LIN {X -32.603,Y -13.521,Z -185.543,A -90.000,B 90.000,C 0.000} C_DIS
LIN {X -30.435,Y -13.512,Z -183.855,A -90.000,B 90.000,C 0.000} C_DIS
LIN {X -29.679,Y -13.512,Z -183.226,A -90.000,B 90.000,C 0.000} C_DIS
LIN {X -27.830,Y -13.506,Z -181.704,A -90.000,B 90.000,C 0.000} C_DIS
LIN {X -27.727,Y -13.503,Z -181.618,A -90.000,B 90.000,C 0.000} C_DIS
LIN {X -27.071,Y -13.503,Z -181.033,A -90.000,B 90.000,C 0.000} C_DIS
LIN {X -25.521,Y -13.499,Z -179.663,A -90.000,B 90.000,C 0.000} C_DIS
LIN {X -25.407,Y -13.501,Z -179.554,A -90.000,B 90.000,C 0.000} C_DIS
LIN {X -24.304,Y -13.500,Z -178.492,A -90.000,B 90.000,C 0.000} C_DIS
LIN {X -23.268,Y -13.500,Z -177.491,A -90.000,B 90.000,C 0.000} C_DIS
LIN {X -23.207,Y -13.501,Z -177.427,A -90.000,B 90.000,C 0.000} C_DIS
LIN {X -21.361,Y -13.502,Z -175.457,A -90.000,B 90.000,C 0.000} C_DIS
LIN {X -21.188,Y -13.509,Z -175.253,A -90.000,B 90.000,C 0.000} C_DIS
LIN {X -20.282,Y -13.511,Z -174.163,A -90.000,B 90.000,C 0.000} C_DIS
LIN {X -19.571,Y -13.511,Z -173.313,A -90.000,B 90.000,C 0.000} C_DIS
LIN {X -19.406,Y -13.519,Z -173.093,A -90.000,B 90.000,C 0.000} C_DIS
LIN {X -18.419,Y -13.525,Z -171.738,A -90.000,B 90.000,C 0.000} C_DIS
LIN {X -17.952,Y -13.526,Z -171.102,A -90.000,B 90.000,C 0.000} C_DIS
LIN {X -17.711,Y -13.540,Z -170.731,A -90.000,B 90.000,C 0.000} C_DIS
LIN {X -16.556,Y -13.547,Z -168.902,A -90.000,B 90.000,C 0.000} C_DIS
LIN {X -16.311,Y -13.564,Z -168.458,A -90.000,B 90.000,C 0.000} C_DIS
LIN {X -16.047,Y -13.566,Z -167.961,A -90.000,B 90.000,C 0.000} C_DIS
LIN {X -15.282,Y -13.568,Z -166.533,A -90.000,B 90.000,C 0.000} C_DIS
LIN {X -15.138,Y -13.584,Z -166.208,A -90.000,B 90.000,C 0.000} C_DIS
LIN {X -14.825,Y -13.585,Z -165.451,A -90.000,B 90.000,C 0.000} C_DIS
LIN {X -14.427,Y -13.582,Z -164.520,A -90.000,B 90.000,C 0.000} C_DIS
LIN {X -14.392,Y -13.581,Z -164.436,A -90.000,B 90.000,C 0.000} C_DIS
LIN {X -14.317,Y -13.597,Z -164.189,A -90.000,B 90.000,C 0.000} C_DIS
LIN {X -14.106,Y -13.597,Z -163.384,A -90.000,B 90.000,C 0.000} C_DIS
LIN {X -13.966,Y -13.591,Z -162.892,A -90.000,B 90.000,C 0.000} C_DIS
LIN {X -13.957,Y -13.602,Z -162.791,A -90.000,B 90.000,C 0.000} C_DIS
LIN {X -13.942,Y -13.600,Z -162.270,A -90.000,B 90.000,C 0.000} C_DIS
LIN {X -13.935,Y -13.598,Z -162.168,A -90.000,B 90.000,C 0.000} C_DIS
LIN {X -13.934,Y -13.580,Z -162.042,A -90.000,B 90.000,C 0.000} C_DIS
LIN {X -13.984,Y -13.577,Z -161.815,A -90.000,B 90.000,C 0.000} C_DIS
LIN {X -14.013,Y -13.564,Z -161.709,A -90.000,B 90.000,C 0.000} C_DIS
LIN {X -14.062,Y -13.537,Z -161.501,A -90.000,B 90.000,C 0.000} C_DIS
LIN {X -14.184,Y -13.531,Z -161.236,A -90.000,B 90.000,C 0.000} C_DIS
LIN {X -14.310,Y -13.506,Z -160.958,A -90.000,B 90.000,C 0.000} C_DIS
LIN {X -14.353,Y -13.506,Z -160.895,A -90.000,B 90.000,C 0.000} C_DIS
LIN {X -14.579,Y -13.497,Z -160.535,A -90.000,B 90.000,C 0.000} C_DIS
LIN {X -14.712,Y -13.489,Z -160.310,A -90.000,B 90.000,C 0.000} C_DIS
LIN {X -14.861,Y -13.476,Z -160.060,A -90.000,B 90.000,C 0.000} C_DIS
LIN {X -15.055,Y -13.476,Z -159.798,A -90.000,B 90.000,C 0.000} C_DIS
LIN {X -15.472,Y -13.453,Z -159.139,A -90.000,B 90.000,C 0.000} C_DIS
LIN {X -15.551,Y -13.447,Z -159.015,A -90.000,B 90.000,C 0.000} C_DIS
LIN {X -15.947,Y -13.442,Z -158.519,A -90.000,B 90.000,C 0.000} C_DIS
LIN {X -16.007,Y -13.439,Z -158.438,A -90.000,B 90.000,C 0.000} C_DIS
LIN {X -16.332,Y -13.428,Z -157.993,A -90.000,B 90.000,C 0.000} C_DIS
LIN {X -16.463,Y -13.420,Z -157.815,A -90.000,B 90.000,C 0.000} C_DIS
LIN {X -16.798,Y -13.420,Z -157.455,A -90.000,B 90.000,C 0.000} C_DIS
LIN {X -17.768,Y -13.398,Z -156.310,A -90.000,B 90.000,C 0.000} C_DIS
LIN {X -18.375,Y -13.398,Z -155.715,A -90.000,B 90.000,C 0.000} C_DIS
LIN {X -19.637,Y -13.380,Z -154.392,A -90.000,B 90.000,C 0.000} C_DIS
LIN {X -20.180,Y -13.380,Z -153.893,A -90.000,B 90.000,C 0.000} C_DIS
LIN {X -20.760,Y -13.378,Z -153.350,A -90.000,B 90.000,C 0.000} C_DIS
LIN {X -22.310,Y -13.366,Z -151.859,A -90.000,B 90.000,C 0.000} C_DIS
LIN {X -23.609,Y -13.366,Z -150.629,A -90.000,B 90.000,C 0.000} C_DIS
LIN {X -25.479,Y -13.356,Z -148.794,A -90.000,B 90.000,C 0.000} C_DIS
LIN {X -26.748,Y -13.355,Z -147.476,A -90.000,B 90.000,C 0.000} C_DIS
LIN {X -28.620,Y -13.347,Z -145.475,A -90.000,B 90.000,C 0.000} C_DIS
LIN {X -29.056,Y -13.347,Z -145.002,A -90.000,B 90.000,C 0.000} C_DIS
LIN {X -30.297,Y -13.346,Z -143.489,A -90.000,B 90.000,C 0.000} C_DIS
LIN {X -32.094,Y -13.341,Z -141.253,A -90.000,B 90.000,C 0.000} C_DIS
LIN {X -32.381,Y -13.341,Z -140.865,A -90.000,B 90.000,C 0.000} C_DIS
LIN {X -33.757,Y -13.338,Z -138.675,A -90.000,B 90.000,C 0.000} C_DIS
LIN {X -34.921,Y -13.339,Z -136.852,A -90.000,B 90.000,C 0.000} C_DIS
LIN {X -34.999,Y -13.339,Z -136.727,A -90.000,B 90.000,C 0.000} C_DIS
LIN {X -35.167,Y -13.339,Z -136.437,A -90.000,B 90.000,C 0.000} C_DIS
LIN {X -36.167,Y -13.338,Z -134.508,A -90.000,B 90.000,C 0.000} C_DIS
LIN {X -37.313,Y -13.340,Z -132.316,A -90.000,B 90.000,C 0.000} C_DIS
LIN {X -38.973,Y -13.342,Z -128.621,A -90.000,B 90.000,C 0.000} C_DIS
LIN {X -39.115,Y -13.342,Z -128.298,A -90.000,B 90.000,C 0.000} C_DIS
LIN {X -39.395,Y -13.342,Z -127.621,A -90.000,B 90.000,C 0.000} C_DIS
LIN {X -40.348,Y -13.344,Z -125.295,A -90.000,B 90.000,C 0.000} C_DIS
LIN {X -40.910,Y -13.345,Z -123.941,A -90.000,B 90.000,C 0.000} C_DIS
LIN {X -41.363,Y -13.344,Z -122.840,A -90.000,B 90.000,C 0.000} C_DIS
LIN {X -41.408,Y -13.345,Z -122.740,A -90.000,B 90.000,C 0.000} C_DIS
LIN {X -42.021,Y -13.344,Z -121.412,A -90.000,B 90.000,C 0.000} C_DIS
LIN {X -42.220,Y -13.344,Z -121.068,A -90.000,B 90.000,C 0.000} C_DIS
LIN {X -42.544,Y -13.344,Z -120.503,A -90.000,B 90.000,C 0.000} C_DIS
LIN {X -42.768,Y -13.341,Z -120.111,A -90.000,B 90.000,C 0.000} C_DIS
LIN {X -43.249,Y -13.341,Z -119.434,A -90.000,B 90.000,C 0.000} C_DIS
LIN {X -43.827,Y -13.338,Z -118.612,A -90.000,B 90.000,C 0.000} C_DIS
LIN {X -44.350,Y -13.336,Z -117.951,A -90.000,B 90.000,C 0.000} C_DIS
LIN {X -45.457,Y -13.336,Z -116.575,A -90.000,B 90.000,C 0.000} C_DIS
LIN {X -45.977,Y -13.336,Z -115.946,A -90.000,B 90.000,C 0.000} C_DIS
LIN {X -47.617,Y -13.336,Z -113.985,A -90.000,B 90.000,C 0.000} C_DIS
LIN {X -49.027,Y -13.339,Z -112.291,A -90.000,B 90.000,C 0.000} C_DIS
LIN {X -50.026,Y -13.341,Z -111.084,A -90.000,B 90.000,C 0.000} C_DIS
LIN {X -50.281,Y -13.340,Z -110.764,A -90.000,B 90.000,C 0.000} C_DIS
LIN {X -52.533,Y -13.344,Z -107.943,A -90.000,B 90.000,C 0.000} C_DIS
LIN {X -52.855,Y -13.342,Z -107.513,A -90.000,B 90.000,C 0.000} C_DIS
LIN {X -55.167,Y -13.345,Z -104.411,A -90.000,B 90.000,C 0.000} C_DIS
LIN {X -55.603,Y -13.344,Z -103.815,A -90.000,B 90.000,C 0.000} C_DIS
LIN {X -57.294,Y -13.348,Z -101.483,A -90.000,B 90.000,C 0.000} C_DIS
LIN {X -59.765,Y -13.350,Z -98.084,A -90.000,B 90.000,C 0.000} C_DIS
LIN {X -60.223,Y -13.354,Z -97.489,A -90.000,B 90.000,C 0.000} C_DIS
LIN {X -60.710,Y -13.355,Z -96.856,A -90.000,B 90.000,C 0.000} C_DIS
LIN {X -61.855,Y -13.356,Z -95.344,A -90.000,B 90.000,C 0.000} C_DIS
LIN {X -62.279,Y -13.365,Z -94.849,A -90.000,B 90.000,C 0.000} C_DIS
LIN {X -63.691,Y -13.370,Z -93.147,A -90.000,B 90.000,C 0.000} C_DIS
LIN {X -64.265,Y -13.390,Z -92.547,A -90.000,B 90.000,C 0.000} C_DIS
LIN {X -64.328,Y -13.392,Z -92.479,A -90.000,B 90.000,C 0.000} C_DIS
LIN {X -65.247,Y -13.396,Z -91.482,A -90.000,B 90.000,C 0.000} C_DIS
LIN {X -65.559,Y -13.400,Z -91.142,A -90.000,B 90.000,C 0.000} C_DIS
LIN {X -65.914,Y -13.415,Z -90.804,A -90.000,B 90.000,C 0.000} C_DIS
LIN {X -66.131,Y -13.423,Z -90.598,A -90.000,B 90.000,C 0.000} C_DIS
LIN {X -66.838,Y -13.428,Z -89.918,A -90.000,B 90.000,C 0.000} C_DIS
LIN {X -67.329,Y -13.437,Z -89.441,A -90.000,B 90.000,C 0.000} C_DIS
LIN {X -67.529,Y -13.448,Z -89.273,A -90.000,B 90.000,C 0.000} C_DIS
LIN {X -67.776,Y -13.460,Z -89.058,A -90.000,B 90.000,C 0.000} C_DIS
LIN {X -68.839,Y -13.470,Z -88.148,A -90.000,B 90.000,C 0.000} C_DIS
LIN {X -69.143,Y -13.476,Z -87.885,A -90.000,B 90.000,C 0.000} C_DIS
LIN {X -69.710,Y -13.502,Z -87.438,A -90.000,B 90.000,C 0.000} C_DIS
LIN {X -70.481,Y -13.518,Z -86.840,A -90.000,B 90.000,C 0.000} C_DIS
LIN {X -71.260,Y -13.526,Z -86.239,A -90.000,B 90.000,C 0.000} C_DIS
LIN {X -71.431,Y -13.531,Z -86.115,A -90.000,B 90.000,C 0.000} C_DIS
LIN {X -72.208,Y -13.546,Z -85.561,A -90.000,B 90.000,C 0.000} C_DIS
LIN {X -73.171,Y -13.557,Z -84.881,A -90.000,B 90.000,C 0.000} C_DIS
LIN {X -73.565,Y -13.567,Z -84.617,A -90.000,B 90.000,C 0.000} C_DIS
LIN {X -74.411,Y -13.579,Z -84.056,A -90.000,B 90.000,C 0.000} C_DIS
LIN {X -75.229,Y -13.585,Z -83.519,A -90.000,B 90.000,C 0.000} C_DIS
LIN {X -75.329,Y -13.587,Z -83.456,A -90.000,B 90.000,C 0.000} C_DIS
LIN {X -77.326,Y -13.585,Z -82.227,A -90.000,B 90.000,C 0.000} C_DIS
LIN {X -77.647,Y -13.579,Z -82.037,A -90.000,B 90.000,C 0.000} C_DIS
LIN {X -78.628,Y -13.564,Z -81.467,A -90.000,B 90.000,C 0.000} C_DIS
LIN {X -78.972,Y -13.556,Z -81.269,A -90.000,B 90.000,C 0.000} C_DIS
LIN {X -79.425,Y -13.542,Z -81.001,A -90.000,B 90.000,C 0.000} C_DIS
LIN {X -79.841,Y -13.533,Z -80.762,A -90.000,B 90.000,C 0.000} C_DIS
LIN {X -80.581,Y -13.519,Z -80.336,A -90.000,B 90.000,C 0.000} C_DIS
LIN {X -81.066,Y -13.502,Z -80.031,A -90.000,B 90.000,C 0.000} C_DIS
LIN {X -81.880,Y -13.483,Z -79.540,A -90.000,B 90.000,C 0.000} C_DIS
LIN {X -82.269,Y -13.469,Z -79.285,A -90.000,B 90.000,C 0.000} C_DIS
LIN {X -82.365,Y -13.465,Z -79.218,A -90.000,B 90.000,C 0.000} C_DIS
LIN {X -83.021,Y -13.449,Z -78.754,A -90.000,B 90.000,C 0.000} C_DIS
LIN {X -83.435,Y -13.442,Z -78.474,A -90.000,B 90.000,C 0.000} C_DIS
LIN {X -83.940,Y -13.424,Z -78.085,A -90.000,B 90.000,C 0.000} C_DIS
LIN {X -84.133,Y -13.420,Z -77.934,A -90.000,B 90.000,C 0.000} C_DIS
LIN {X -84.397,Y -13.417,Z -77.725,A -90.000,B 90.000,C 0.000} C_DIS
LIN {X -84.820,Y -13.410,Z -77.380,A -90.000,B 90.000,C 0.000} C_DIS
LIN {X -85.096,Y -13.403,Z -77.146,A -90.000,B 90.000,C 0.000} C_DIS
LIN {X -85.559,Y -13.396,Z -76.749,A -90.000,B 90.000,C 0.000} C_DIS
LIN {X -86.655,Y -13.387,Z -75.802,A -90.000,B 90.000,C 0.000} C_DIS
LIN {X -87.183,Y -13.390,Z -75.370,A -90.000,B 90.000,C 0.000} C_DIS
LIN {X -87.545,Y -13.402,Z -75.116,A -90.000,B 90.000,C 0.000} C_DIS
LIN {X -87.805,Y -13.409,Z -74.928,A -90.000,B 90.000,C 0.000} C_DIS
LIN {X -88.004,Y -13.420,Z -74.806,A -90.000,B 90.000,C 0.000} C_DIS
LIN {X -88.411,Y -13.437,Z -74.558,A -90.000,B 90.000,C 0.000} C_DIS
LIN {X -88.591,Y -13.446,Z -74.444,A -90.000,B 90.000,C 0.000} C_DIS
LIN {X -88.766,Y -13.458,Z -74.347,A -90.000,B 90.000,C 0.000} C_DIS
LIN {X -89.213,Y -13.480,Z -74.105,A -90.000,B 90.000,C 0.000} C_DIS
LIN {X -89.470,Y -13.502,Z -73.977,A -90.000,B 90.000,C 0.000} C_DIS
LIN {X -89.913,Y -13.524,Z -73.765,A -90.000,B 90.000,C 0.000} C_DIS
LIN {X -90.100,Y -13.530,Z -73.677,A -90.000,B 90.000,C 0.000} C_DIS
LIN {X -90.481,Y -13.548,Z -73.514,A -90.000,B 90.000,C 0.000} C_DIS
LIN {X -90.587,Y -13.548,Z -73.470,A -90.000,B 90.000,C 0.000} C_DIS
LIN {X -90.887,Y -13.556,Z -73.360,A -90.000,B 90.000,C 0.000} C_DIS
LIN {X -91.237,Y -13.568,Z -73.226,A -90.000,B 90.000,C 0.000} C_DIS
LIN {X -91.807,Y -13.585,Z -73.041,A -90.000,B 90.000,C 0.000} C_DIS
LIN {X -92.036,Y -13.588,Z -72.964,A -90.000,B 90.000,C 0.000} C_DIS
LIN {X -92.265,Y -13.597,Z -72.896,A -90.000,B 90.000,C 0.000} C_DIS
LIN {X -92.393,Y -13.601,Z -72.858,A -90.000,B 90.000,C 0.000} C_DIS
LIN {X -92.838,Y -13.609,Z -72.737,A -90.000,B 90.000,C 0.000} C_DIS
LIN {X -93.306,Y -13.628,Z -72.603,A -90.000,B 90.000,C 0.000} C_DIS
LIN {X -93.442,Y -13.639,Z -72.572,A -90.000,B 90.000,C 0.000} C_DIS
LIN {X -93.652,Y -13.647,Z -72.528,A -90.000,B 90.000,C 0.000} C_DIS
LIN {X -94.040,Y -13.653,Z -72.428,A -90.000,B 90.000,C 0.000} C_DIS
LIN {X -94.194,Y -13.660,Z -72.396,A -90.000,B 90.000,C 0.000} C_DIS
LIN {X -94.571,Y -13.685,Z -72.310,A -90.000,B 90.000,C 0.000} C_DIS
LIN {X -94.679,Y -13.686,Z -72.289,A -90.000,B 90.000,C 0.000} C_DIS
LIN {X -94.926,Y -13.698,Z -72.235,A -90.000,B 90.000,C 0.000} C_DIS
LIN {X -95.117,Y -13.701,Z -72.204,A -90.000,B 90.000,C 0.000} C_DIS
LIN {X -95.405,Y -13.697,Z -72.146,A -90.000,B 90.000,C 0.000} C_DIS
LIN {X -95.701,Y -13.700,Z -72.080,A -90.000,B 90.000,C 0.000} C_DIS
LIN {X -95.954,Y -13.707,Z -72.021,A -90.000,B 90.000,C 0.000} C_DIS
LIN {X -96.385,Y -13.716,Z -71.912,A -90.000,B 90.000,C 0.000} C_DIS
LIN {X -96.673,Y -13.714,Z -71.830,A -90.000,B 90.000,C 0.000} C_DIS
LIN {X -97.041,Y -13.735,Z -71.751,A -90.000,B 90.000,C 0.000} C_DIS
LIN {X -97.161,Y -13.738,Z -71.720,A -90.000,B 90.000,C 0.000} C_DIS
LIN {X -97.475,Y -13.755,Z -71.632,A -90.000,B 90.000,C 0.000} C_DIS
LIN {X -97.556,Y -13.755,Z -71.603,A -90.000,B 90.000,C 0.000} C_DIS
LIN {X -97.746,Y -13.742,Z -71.544,A -90.000,B 90.000,C 0.000} C_DIS
LIN {X -97.820,Y -13.742,Z -71.524,A -90.000,B 90.000,C 0.000} C_DIS
LIN {X -98.228,Y -13.745,Z -71.409,A -90.000,B 90.000,C 0.000} C_DIS
LIN {X -98.319,Y -13.748,Z -71.382,A -90.000,B 90.000,C 0.000} C_DIS
LIN {X -98.620,Y -13.766,Z -71.278,A -90.000,B 90.000,C 0.000} C_DIS
LIN {X -98.739,Y -13.769,Z -71.232,A -90.000,B 90.000,C 0.000} C_DIS
LIN {X -99.031,Y -13.763,Z -71.127,A -90.000,B 90.000,C 0.000} C_DIS
LIN {X -99.176,Y -13.751,Z -71.064,A -90.000,B 90.000,C 0.000} C_DIS
LIN {X -99.293,Y -13.747,Z -71.019,A -90.000,B 90.000,C 0.000} C_DIS
LIN {X -99.392,Y -13.745,Z -70.979,A -90.000,B 90.000,C 0.000} C_DIS
LIN {X -99.879,Y -13.747,Z -70.774,A -90.000,B 90.000,C 0.000} C_DIS
LIN {X -100.025,Y -13.753,Z -70.708,A -90.000,B 90.000,C 0.000} C_DIS
LIN {X -100.169,Y -13.762,Z -70.638,A -90.000,B 90.000,C 0.000} C_DIS
LIN {X -100.225,Y -13.764,Z -70.613,A -90.000,B 90.000,C 0.000} C_DIS
LIN {X -100.408,Y -13.763,Z -70.523,A -90.000,B 90.000,C 0.000} C_DIS
LIN {X -100.626,Y -13.760,Z -70.412,A -90.000,B 90.000,C 0.000} C_DIS
LIN {X -100.877,Y -13.742,Z -70.265,A -90.000,B 90.000,C 0.000} C_DIS
LIN {X -101.019,Y -13.735,Z -70.186,A -90.000,B 90.000,C 0.000} C_DIS
LIN {X -101.099,Y -13.732,Z -70.139,A -90.000,B 90.000,C 0.000} C_DIS
LIN {X -101.550,Y -13.728,Z -69.870,A -90.000,B 90.000,C 0.000} C_DIS
LIN {X -101.664,Y -13.731,Z -69.798,A -90.000,B 90.000,C 0.000} C_DIS
LIN {X -101.861,Y -13.742,Z -69.669,A -90.000,B 90.000,C 0.000} C_DIS
LIN {X -101.983,Y -13.747,Z -69.586,A -90.000,B 90.000,C 0.000} C_DIS
LIN {X -102.253,Y -13.751,Z -69.404,A -90.000,B 90.000,C 0.000} C_DIS
LIN {X -102.723,Y -13.726,Z -69.039,A -90.000,B 90.000,C 0.000} C_DIS
LIN {X -103.242,Y -13.708,Z -68.624,A -90.000,B 90.000,C 0.000} C_DIS
LIN {X -103.469,Y -13.715,Z -68.430,A -90.000,B 90.000,C 0.000} C_DIS
LIN {X -103.893,Y -13.722,Z -68.046,A -90.000,B 90.000,C 0.000} C_DIS
LIN {X -104.288,Y -13.712,Z -67.655,A -90.000,B 90.000,C 0.000} C_DIS
LIN {X -104.740,Y -13.708,Z -67.195,A -90.000,B 90.000,C 0.000} C_DIS
LIN {X -104.913,Y -13.705,Z -67.016,A -90.000,B 90.000,C 0.000} C_DIS
LIN {X -105.275,Y -13.712,Z -66.623,A -90.000,B 90.000,C 0.000} C_DIS
LIN {X -105.486,Y -13.721,Z -66.390,A -90.000,B 90.000,C 0.000} C_DIS
LIN {X -105.650,Y -13.724,Z -66.200,A -90.000,B 90.000,C 0.000} C_DIS
LIN {X -106.104,Y -13.721,Z -65.650,A -90.000,B 90.000,C 0.000} C_DIS
LIN {X -106.183,Y -13.718,Z -65.550,A -90.000,B 90.000,C 0.000} C_DIS
LIN {X -106.477,Y -13.721,Z -65.165,A -90.000,B 90.000,C 0.000} C_DIS
LIN {X -106.683,Y -13.733,Z -64.882,A -90.000,B 90.000,C 0.000} C_DIS
LIN {X -106.951,Y -13.751,Z -64.500,A -90.000,B 90.000,C 0.000} C_DIS
LIN {X -107.337,Y -13.769,Z -63.915,A -90.000,B 90.000,C 0.000} C_DIS
LIN {X -107.580,Y -13.784,Z -63.538,A -90.000,B 90.000,C 0.000} C_DIS
LIN {X -107.987,Y -13.814,Z -62.895,A -90.000,B 90.000,C 0.000} C_DIS
LIN {X -108.225,Y -13.831,Z -62.481,A -90.000,B 90.000,C 0.000} C_DIS
LIN {X -108.561,Y -13.845,Z -61.866,A -90.000,B 90.000,C 0.000} C_DIS
LIN {X -108.601,Y -13.848,Z -61.791,A -90.000,B 90.000,C 0.000} C_DIS
LIN {X -108.850,Y -13.867,Z -61.247,A -90.000,B 90.000,C 0.000} C_DIS
LIN {X -108.900,Y -13.870,Z -61.134,A -90.000,B 90.000,C 0.000} C_DIS
LIN {X -108.965,Y -13.872,Z -60.978,A -90.000,B 90.000,C 0.000} C_DIS
LIN {X -109.188,Y -13.886,Z -60.425,A -90.000,B 90.000,C 0.000} C_DIS
LIN {X -109.273,Y -13.892,Z -60.203,A -90.000,B 90.000,C 0.000} C_DIS
LIN {X -109.480,Y -13.908,Z -59.653,A -90.000,B 90.000,C 0.000} C_DIS
LIN {X -109.572,Y -13.912,Z -59.383,A -90.000,B 90.000,C 0.000} C_DIS
LIN {X -109.688,Y -13.925,Z -59.019,A -90.000,B 90.000,C 0.000} C_DIS
LIN {X -109.730,Y -13.924,Z -58.867,A -90.000,B 90.000,C 0.000} C_DIS
LIN {X -109.928,Y -13.928,Z -58.109,A -90.000,B 90.000,C 0.000} C_DIS
LIN {X -110.035,Y -13.920,Z -57.624,A -90.000,B 90.000,C 0.000} C_DIS
LIN {X -110.116,Y -13.914,Z -57.247,A -90.000,B 90.000,C 0.000} C_DIS
LIN {X -110.131,Y -13.905,Z -57.213,A -90.000,B 90.000,C 0.000} C_DIS
LIN {X -110.346,Y -13.789,Z -56.721,A -90.000,B 90.000,C 0.000} C_DIS
LIN {X -110.434,Y -13.743,Z -56.509,A -90.000,B 90.000,C 0.000} C_DIS
LIN {X -110.484,Y -13.712,Z -56.379,A -90.000,B 90.000,C 0.000} C_DIS
LIN {X -110.575,Y -13.661,Z -56.147,A -90.000,B 90.000,C 0.000} C_DIS
LIN {X -110.656,Y -13.613,Z -55.927,A -90.000,B 90.000,C 0.000} C_DIS
LIN {X -110.705,Y -13.586,Z -55.780,A -90.000,B 90.000,C 0.000} C_DIS
LIN {X -110.762,Y -13.559,Z -55.621,A -90.000,B 90.000,C 0.000} C_DIS
LIN {X -110.902,Y -13.484,Z -55.162,A -90.000,B 90.000,C 0.000} C_DIS
LIN {X -110.945,Y -13.468,Z -55.041,A -90.000,B 90.000,C 0.000} C_DIS
LIN {X -111.038,Y -13.436,Z -54.756,A -90.000,B 90.000,C 0.000} C_DIS
LIN {X -111.059,Y -13.428,Z -54.684,A -90.000,B 90.000,C 0.000} C_DIS
LIN {X -111.158,Y -13.405,Z -54.413,A -90.000,B 90.000,C 0.000} C_DIS
LIN {X -111.204,Y -13.396,Z -54.293,A -90.000,B 90.000,C 0.000} C_DIS
LIN {X -111.326,Y -13.402,Z -54.128,A -90.000,B 90.000,C 0.000} C_DIS
LIN {X -111.517,Y -13.408,Z -53.852,A -90.000,B 90.000,C 0.000} C_DIS
LIN {X -111.684,Y -13.419,Z -53.601,A -90.000,B 90.000,C 0.000} C_DIS
LIN {X -111.889,Y -13.434,Z -53.283,A -90.000,B 90.000,C 0.000} C_DIS
LIN {X -112.098,Y -13.450,Z -52.934,A -90.000,B 90.000,C 0.000} C_DIS
LIN {X -112.252,Y -13.460,Z -52.632,A -90.000,B 90.000,C 0.000} C_DIS
LIN {X -112.393,Y -13.472,Z -52.351,A -90.000,B 90.000,C 0.000} C_DIS
LIN {X -112.504,Y -13.484,Z -52.105,A -90.000,B 90.000,C 0.000} C_DIS
LIN {X -112.601,Y -13.494,Z -51.879,A -90.000,B 90.000,C 0.000} C_DIS
LIN {X -112.646,Y -13.500,Z -51.769,A -90.000,B 90.000,C 0.000} C_DIS
LIN {X -112.707,Y -13.514,Z -51.618,A -90.000,B 90.000,C 0.000} C_DIS
LIN {X -112.754,Y -13.524,Z -51.494,A -90.000,B 90.000,C 0.000} C_DIS
LIN {X -112.890,Y -13.549,Z -51.073,A -90.000,B 90.000,C 0.000} C_DIS
LIN {X -112.921,Y -13.553,Z -50.961,A -90.000,B 90.000,C 0.000} C_DIS
LIN {X -112.997,Y -13.572,Z -50.659,A -90.000,B 90.000,C 0.000} C_DIS
LIN {X -113.031,Y -13.581,Z -50.515,A -90.000,B 90.000,C 0.000} C_DIS
LIN {X -113.098,Y -13.601,Z -50.221,A -90.000,B 90.000,C 0.000} C_DIS
LIN {X -113.154,Y -13.618,Z -49.918,A -90.000,B 90.000,C 0.000} C_DIS
LIN {X -113.169,Y -13.625,Z -49.829,A -90.000,B 90.000,C 0.000} C_DIS
LIN {X -113.178,Y -13.632,Z -49.767,A -90.000,B 90.000,C 0.000} C_DIS
LIN {X -113.204,Y -13.655,Z -49.352,A -90.000,B 90.000,C 0.000} C_DIS
LIN {X -113.216,Y -13.675,Z -49.060,A -90.000,B 90.000,C 0.000} C_DIS
LIN {X -113.223,Y -13.722,Z -48.612,A -90.000,B 90.000,C 0.000} C_DIS
LIN {X -113.194,Y -13.750,Z -48.192,A -90.000,B 90.000,C 0.000} C_DIS
LIN {X -113.175,Y -13.752,Z -48.059,A -90.000,B 90.000,C 0.000} C_DIS
LIN {X -113.144,Y -13.761,Z -47.877,A -90.000,B 90.000,C 0.000} C_DIS
LIN {X -113.074,Y -13.785,Z -47.489,A -90.000,B 90.000,C 0.000} C_DIS
LIN {X -113.007,Y -13.817,Z -47.182,A -90.000,B 90.000,C 0.000} C_DIS
LIN {X -112.959,Y -13.824,Z -47.019,A -90.000,B 90.000,C 0.000} C_DIS
LIN {X -112.853,Y -13.845,Z -46.677,A -90.000,B 90.000,C 0.000} C_DIS
LIN {X -112.816,Y -13.849,Z -46.568,A -90.000,B 90.000,C 0.000} C_DIS
LIN {X -112.766,Y -13.858,Z -46.429,A -90.000,B 90.000,C 0.000} C_DIS
LIN {X -112.648,Y -13.870,Z -46.151,A -90.000,B 90.000,C 0.000} C_DIS
LIN {X -112.651,Y -13.778,Z -45.920,A -90.000,B 90.000,C 0.000} C_DIS
LIN {X -112.644,Y -13.689,Z -45.670,A -90.000,B 90.000,C 0.000} C_DIS
LIN {X -112.638,Y -13.656,Z -45.571,A -90.000,B 90.000,C 0.000} C_DIS
LIN {X -112.625,Y -13.605,Z -45.413,A -90.000,B 90.000,C 0.000} C_DIS
LIN {X -112.611,Y -13.569,Z -45.301,A -90.000,B 90.000,C 0.000} C_DIS
LIN {X -112.581,Y -13.514,Z -45.123,A -90.000,B 90.000,C 0.000} C_DIS
LIN {X -112.550,Y -13.470,Z -44.963,A -90.000,B 90.000,C 0.000} C_DIS
LIN {X -112.622,Y -13.473,Z -44.815,A -90.000,B 90.000,C 0.000} C_DIS
LIN {X -112.766,Y -13.478,Z -44.510,A -90.000,B 90.000,C 0.000} C_DIS
LIN {X -113.073,Y -13.490,Z -43.847,A -90.000,B 90.000,C 0.000} C_DIS
LIN {X -113.204,Y -13.502,Z -43.553,A -90.000,B 90.000,C 0.000} C_DIS
LIN {X -113.296,Y -13.510,Z -43.328,A -90.000,B 90.000,C 0.000} C_DIS
LIN {X -113.422,Y -13.519,Z -43.003,A -90.000,B 90.000,C 0.000} C_DIS
LIN {X -113.481,Y -13.522,Z -42.832,A -90.000,B 90.000,C 0.000} C_DIS
LIN {X -113.639,Y -13.538,Z -42.362,A -90.000,B 90.000,C 0.000} C_DIS
LIN {X -113.726,Y -13.552,Z -42.092,A -90.000,B 90.000,C 0.000} C_DIS
LIN {X -113.746,Y -13.554,Z -42.022,A -90.000,B 90.000,C 0.000} C_DIS
LIN {X -113.966,Y -13.586,Z -41.233,A -90.000,B 90.000,C 0.000} C_DIS
LIN {X -114.008,Y -13.590,Z -41.055,A -90.000,B 90.000,C 0.000} C_DIS
LIN {X -114.065,Y -13.602,Z -40.776,A -90.000,B 90.000,C 0.000} C_DIS
LIN {X -114.144,Y -13.624,Z -40.346,A -90.000,B 90.000,C 0.000} C_DIS
LIN {X -114.174,Y -13.633,Z -40.141,A -90.000,B 90.000,C 0.000} C_DIS
LIN {X -114.195,Y -13.643,Z -39.982,A -90.000,B 90.000,C 0.000} C_DIS
LIN {X -114.209,Y -13.648,Z -39.813,A -90.000,B 90.000,C 0.000} C_DIS
LIN {X -114.248,Y -13.682,Z -39.205,A -90.000,B 90.000,C 0.000} C_DIS
LIN {X -114.255,Y -13.690,Z -39.054,A -90.000,B 90.000,C 0.000} C_DIS
LIN {X -114.261,Y -13.700,Z -38.878,A -90.000,B 90.000,C 0.000} C_DIS
LIN {X -114.261,Y -13.707,Z -38.706,A -90.000,B 90.000,C 0.000} C_DIS
LIN {X -114.259,Y -13.715,Z -38.584,A -90.000,B 90.000,C 0.000} C_DIS
LIN {X -114.236,Y -13.737,Z -38.185,A -90.000,B 90.000,C 0.000} C_DIS
LIN {X -114.206,Y -13.752,Z -37.845,A -90.000,B 90.000,C 0.000} C_DIS
LIN {X -114.143,Y -13.768,Z -37.481,A -90.000,B 90.000,C 0.000} C_DIS
LIN {X -114.069,Y -13.789,Z -37.089,A -90.000,B 90.000,C 0.000} C_DIS
LIN {X -114.024,Y -13.792,Z -36.912,A -90.000,B 90.000,C 0.000} C_DIS
LIN {X -113.941,Y -13.800,Z -36.606,A -90.000,B 90.000,C 0.000} C_DIS
LIN {X -113.884,Y -13.810,Z -36.414,A -90.000,B 90.000,C 0.000} C_DIS
LIN {X -113.768,Y -13.819,Z -36.071,A -90.000,B 90.000,C 0.000} C_DIS
LIN {X -113.712,Y -13.820,Z -35.915,A -90.000,B 90.000,C 0.000} C_DIS
LIN {X -113.655,Y -13.824,Z -35.769,A -90.000,B 90.000,C 0.000} C_DIS
LIN {X -113.579,Y -13.831,Z -35.587,A -90.000,B 90.000,C 0.000} C_DIS
LIN {X -113.491,Y -13.841,Z -35.383,A -90.000,B 90.000,C 0.000} C_DIS
LIN {X -113.367,Y -13.849,Z -35.124,A -90.000,B 90.000,C 0.000} C_DIS
LIN {X -113.312,Y -13.850,Z -35.021,A -90.000,B 90.000,C 0.000} C_DIS
LIN {X -113.163,Y -13.859,Z -34.756,A -90.000,B 90.000,C 0.000} C_DIS
LIN {X -113.011,Y -13.871,Z -34.509,A -90.000,B 90.000,C 0.000} C_DIS
LIN {X -112.913,Y -13.870,Z -34.366,A -90.000,B 90.000,C 0.000} C_DIS
LIN {X -112.850,Y -13.872,Z -34.278,A -90.000,B 90.000,C 0.000} C_DIS
LIN {X -112.767,Y -13.877,Z -34.165,A -90.000,B 90.000,C 0.000} C_DIS
LIN {X -112.668,Y -13.880,Z -34.036,A -90.000,B 90.000,C 0.000} C_DIS
LIN {X -112.584,Y -13.886,Z -33.929,A -90.000,B 90.000,C 0.000} C_DIS
LIN {X -112.393,Y -13.886,Z -33.712,A -90.000,B 90.000,C 0.000} C_DIS
LIN {X -112.303,Y -13.888,Z -33.613,A -90.000,B 90.000,C 0.000} C_DIS
LIN {X -112.239,Y -13.891,Z -33.548,A -90.000,B 90.000,C 0.000} C_DIS
LIN {X -112.082,Y -13.898,Z -33.396,A -90.000,B 90.000,C 0.000} C_DIS
